LIN {X 0,Y 224.988,Z 280.423,A -85,B 0,C 180,E1 -22090.658,E2 -22090.658} C_VEL
LIN {X 0,Y 227.045,Z 246.583,A -85,B 0,C 180,E1 -22091.716,E2 -22091.716} C_VEL
LIN {X 0,Y 226.588,Z 244.432,A -85,B 0,C 180,E1 -22091.955,E2 -22091.955} C_VEL
LIN {X 0,Y 221.706,Z 232.717,A -85,B 0,C 180,E1 -22094.047,E2 -22094.047} C_VEL
LIN {X 0,Y 216.446,Z 222.08,A -85,B 0,C 180,E1 -22096.416,E2 -22096.416} C_VEL
LIN {X 0,Y 211.273,Z 212.801,A -85,B 0,C 180,E1 -22098.988,E2 -22098.988} C_VEL
LIN {X 0,Y 207.639,Z 206.885,A -85,B 0,C 180,E1 -22100.948,E2 -22100.948} C_VEL
LIN {X 0,Y 204.559,Z 201.986,A -85,B 0,C 180,E1 -22102.75,E2 -22102.75} C_VEL
LIN {X 0,Y 200.929,Z 196.512,A -85,B 0,C 180,E1 -22105.098,E2 -22105.098} C_VEL
LIN {X 0,Y 196.507,Z 190.274,A -85,B 0,C 180,E1 -22108.383,E2 -22108.383} C_VEL
LIN {X 0,Y 192.458,Z 184.954,A -85,B 0,C 180,E1 -22111.954,E2 -22111.954} C_VEL
LIN {X 0,Y 191.731,Z 183.77,A -85,B 0,C 180,E1 -22112.728,E2 -22112.728} C_VEL
LIN {X 0,Y 188.179,Z 179.993,A -85,B 0,C 180,E1 -22116.911,E2 -22116.911} C_VEL
LIN {X 0,Y 186.22,Z 177.647,A -85,B 0,C 180,E1 -22119.999,E2 -22119.999} C_VEL
LIN {X 0,Y 185.766,Z 176.032,A -85,B 0,C 180,E1 -22121.256,E2 -22121.256} C_VEL
LIN {X 0,Y 185.661,Z 175.348,A -85,B 0,C 180,E1 -22123.505,E2 -22123.505} C_VEL
LIN {X 0,Y 185.889,Z 175.33,A -85,B 0,C 180,E1 -22129.418,E2 -22129.418} C_VEL
LIN {X 0,Y 185.931,Z 175.314,A -85,B 0,C 180,E1 -22133.488,E2 -22133.488} C_VEL
LIN {X 0,Y 186.178,Z 175.278,A -85,B 0,C 180,E1 -22137.835,E2 -22137.835} C_VEL
LIN {X 0,Y 186.347,Z 175.263,A -85,B 0,C 180,E1 -22140.269,E2 -22140.269} C_VEL
LIN {X 0,Y 186.866,Z 177.432,A -85,B 0,C 180,E1 -22141.48,E2 -22141.48} C_VEL
LIN {X 0,Y 188.498,Z 179.95,A -85,B 0,C 180,E1 -22144.008,E2 -22144.008} C_VEL
LIN {X 0,Y 191.327,Z 181.512,A -85,B 0,C 180,E1 -22147.166,E2 -22147.166} C_VEL
LIN {X 0,Y 192.658,Z 184.369,A -85,B 0,C 180,E1 -22148.694,E2 -22148.694} C_VEL
LIN {X 0,Y 195.421,Z 186.847,A -85,B 0,C 180,E1 -22151.079,E2 -22151.079} C_VEL
LIN {X 0,Y 196.081,Z 187.718,A -85,B 0,C 180,E1 -22151.63,E2 -22151.63} C_VEL
LIN {X 0,Y 198.151,Z 190.841,A -85,B 0,C 180,E1 -22153.295,E2 -22153.295} C_VEL
LIN {X 0,Y 200.301,Z 192.877,A -85,B 0,C 180,E1 -22154.785,E2 -22154.785} C_VEL
LIN {X 0,Y 202.888,Z 196.511,A -85,B 0,C 180,E1 -22156.531,E2 -22156.531} C_VEL
LIN {X 0,Y 204.322,Z 198.272,A -85,B 0,C 180,E1 -22157.411,E2 -22157.411} C_VEL
LIN {X 0,Y 207.184,Z 201.939,A -85,B 0,C 180,E1 -22159.055,E2 -22159.055} C_VEL
LIN {X 0,Y 211.633,Z 208.287,A -85,B 0,C 180,E1 -22161.424,E2 -22161.424} C_VEL
LIN {X 0,Y 216.087,Z 214.791,A -85,B 0,C 180,E1 -22163.574,E2 -22163.574} C_VEL
LIN {X 0,Y 221.021,Z 223.069,A -85,B 0,C 180,E1 -22165.767,E2 -22165.767} C_VEL
LIN {X 0,Y 226.41,Z 233.873,A -85,B 0,C 180,E1 -22168.017,E2 -22168.017} C_VEL
LIN {X 0,Y 227.763,Z 236.952,A -85,B 0,C 180,E1 -22168.568,E2 -22168.568} C_VEL
LIN {X 0,Y 224.854,Z 278.71,A -85,B 0,C 180,E1 -22169.862,E2 -22169.862} C_VEL
LIN {X 0,Y 222.95,Z 292.239,A -85,B 0,C 180,E1 -22170.585,E2 -22170.585} C_VEL
LIN {X 0,Y 220.678,Z 304.196,A -85,B 0,C 180,E1 -22171.579,E2 -22171.579} C_VEL
LIN {X 0,Y 217.56,Z 315.965,A -85,B 0,C 180,E1 -22172.871,E2 -22172.871} C_VEL
LIN {X 0,Y 214.251,Z 326.305,A -85,B 0,C 180,E1 -22174.361,E2 -22174.361} C_VEL
LIN {X 0,Y 210.299,Z 336.7,A -85,B 0,C 180,E1 -22176.27,E2 -22176.27} C_VEL
LIN {X 0,Y 206.292,Z 345.823,A -85,B 0,C 180,E1 -22178.411,E2 -22178.411} C_VEL
LIN {X 0,Y 201.831,Z 354.704,A -85,B 0,C 180,E1 -22181.104,E2 -22181.104} C_VEL
LIN {X 0,Y 197.677,Z 362.007,A -85,B 0,C 180,E1 -22183.95,E2 -22183.95} C_VEL
LIN {X 0,Y 194.468,Z 367.315,A -85,B 0,C 180,E1 -22186.634,E2 -22186.634} C_VEL
LIN {X 0,Y 191.099,Z 372.35,A -85,B 0,C 180,E1 -22189.941,E2 -22189.941} C_VEL
LIN {X 0,Y 188.379,Z 376.088,A -85,B 0,C 180,E1 -22193.35,E2 -22193.35} C_VEL
LIN {X 0,Y 186.697,Z 378.058,A -85,B 0,C 180,E1 -22195.909,E2 -22195.909} C_VEL
LIN {X 0,Y 185.598,Z 379.226,A -85,B 0,C 180,E1 -22197.986,E2 -22197.986} C_VEL
LIN {X 0,Y 184.271,Z 380.301,A -85,B 0,C 180,E1 -22201.305,E2 -22201.305} C_VEL
LIN {X 0,Y 183.319,Z 380.428,A -85,B 0,C 180,E1 -22205.058,E2 -22205.058} C_VEL
LIN {X 0,Y 183.017,Z 379.943,A -85,B 0,C 180,E1 -22207.418,E2 -22207.418} C_VEL
LIN {X 0,Y 182.831,Z 378.973,A -85,B 0,C 180,E1 -22209.76,E2 -22209.76} C_VEL
LIN {X 0,Y 183.023,Z 376.309,A -85,B 0,C 180,E1 -22213.732,E2 -22213.732} C_VEL
LIN {X 0,Y 183.704,Z 372.053,A -85,B 0,C 180,E1 -22217.854,E2 -22217.854} C_VEL
LIN {X 0,Y 184.693,Z 366.57,A -85,B 0,C 180,E1 -22221.625,E2 -22221.625} C_VEL
LIN {X 0,Y 186.106,Z 359.926,A -85,B 0,C 180,E1 -22225.126,E2 -22225.126} C_VEL
LIN {X 0,Y 187.845,Z 352.004,A -85,B 0,C 180,E1 -22228.392,E2 -22228.392} C_VEL
LIN {X 0,Y 189.79,Z 343.547,A -85,B 0,C 180,E1 -22231.151,E2 -22231.151} C_VEL
LIN {X 0,Y 192.004,Z 333.872,A -85,B 0,C 180,E1 -22233.673,E2 -22233.673} C_VEL
LIN {X 0,Y 194.19,Z 322.773,A -85,B 0,C 180,E1 -22235.973,E2 -22235.973} C_VEL
LIN {X 0,Y 196.122,Z 311.841,A -85,B 0,C 180,E1 -22237.723,E2 -22237.723} C_VEL
LIN {X 0,Y 197.792,Z 299.873,A -85,B 0,C 180,E1 -22239.201,E2 -22239.201} C_VEL
LIN {X 0,Y 199.172,Z 286.973,A -85,B 0,C 180,E1 -22240.355,E2 -22240.355} C_VEL
LIN {X 0,Y 200.126,Z 274.306,A -85,B 0,C 180,E1 -22241.074,E2 -22241.074} C_VEL
LIN {X 0,Y 202.77,Z 214.463,A -85,B 0,C 180,E1 -22243.143,E2 -22243.143} C_VEL
LIN {X 0,Y 198.505,Z 201.646,A -85,B 0,C 180,E1 -22244.291,E2 -22244.291} C_VEL
LIN {X 0,Y 190.934,Z 186.085,A -85,B 0,C 180,E1 -22246.169,E2 -22246.169} C_VEL
LIN {X 0,Y 186.573,Z 178.087,A -85,B 0,C 180,E1 -22247.29,E2 -22247.29} C_VEL
LIN {X 0,Y 185.642,Z 175.362,A -85,B 0,C 180,E1 -22247.63,E2 -22247.63} C_VEL
LIN {X 0,Y 185.535,Z 175.354,A -85,B 0,C 180,E1 -22252.26,E2 -22252.26} C_VEL
LIN {X 0,Y 185.485,Z 175.339,A -85,B 0,C 180,E1 -22257.045,E2 -22257.045} C_VEL
LIN {X 0,Y 185.528,Z 175.375,A -85,B 0,C 180,E1 -22262.029,E2 -22262.029} C_VEL
LIN {X 0,Y 185.497,Z 175.361,A -85,B 0,C 180,E1 -22267.316,E2 -22267.316} C_VEL
LIN {X 0,Y 185.459,Z 175.383,A -85,B 0,C 180,E1 -22270.722,E2 -22270.722} C_VEL
LIN {X 0,Y 185.453,Z 175.353,A -85,B 0,C 180,E1 -22276.058,E2 -22276.058} C_VEL
LIN {X 0,Y 185.455,Z 175.373,A -85,B 0,C 180,E1 -22279.894,E2 -22279.894} C_VEL
LIN {X 0,Y 185.5,Z 175.378,A -85,B 0,C 180,E1 -22282.715,E2 -22282.715} C_VEL
LIN {X 0,Y 185.531,Z 175.345,A -85,B 0,C 180,E1 -22287.974,E2 -22287.974} C_VEL
LIN {X 0,Y 185.547,Z 175.327,A -85,B 0,C 180,E1 -22290.597,E2 -22290.597} C_VEL
LIN {X 0,Y 185.545,Z 175.365,A -85,B 0,C 180,E1 -22295.378,E2 -22295.378} C_VEL
LIN {X 0,Y 185.626,Z 175.356,A -85,B 0,C 180,E1 -22301.18,E2 -22301.18} C_VEL
LIN {X 0,Y 185.698,Z 175.353,A -85,B 0,C 180,E1 -22306.876,E2 -22306.876} C_VEL
LIN {X 0,Y 185.975,Z 175.306,A -85,B 0,C 180,E1 -22311.307,E2 -22311.307} C_VEL
LIN {X 0,Y 186.177,Z 175.29,A -85,B 0,C 180,E1 -22317.838,E2 -22317.838} C_VEL
LIN {X 0,Y 186.383,Z 175.258,A -85,B 0,C 180,E1 -22320.001,E2 -22320.001} C_VEL
LIN {X 0,Y 185.888,Z 175.331,A -85,B 0,C 180,E1 -22324.338,E2 -22324.338} C_VEL
LIN {X 0,Y 185.978,Z 175.309,A -85,B 0,C 180,E1 -22328.695,E2 -22328.695} C_VEL
LIN {X 0,Y 185.711,Z 175.354,A -85,B 0,C 180,E1 -22333.125,E2 -22333.125} C_VEL
LIN {X 0,Y 185.629,Z 175.361,A -85,B 0,C 180,E1 -22338.822,E2 -22338.822} C_VEL
LIN {X 0,Y 185.582,Z 175.368,A -85,B 0,C 180,E1 -22344.647,E2 -22344.647} C_VEL
LIN {X 0,Y 185.548,Z 175.372,A -85,B 0,C 180,E1 -22349.5,E2 -22349.5} C_VEL
LIN {X 0,Y 185.501,Z 175.379,A -85,B 0,C 180,E1 -22354.633,E2 -22354.633} C_VEL
LIN {X 0,Y 185.503,Z 175.38,A -85,B 0,C 180,E1 -22357.315,E2 -22357.315} C_VEL
LIN {X 0,Y 185.465,Z 175.387,A -85,B 0,C 180,E1 -22360.721,E2 -22360.721} C_VEL
LIN {X 0,Y 185.46,Z 175.388,A -85,B 0,C 180,E1 -22366.056,E2 -22366.056} C_VEL
LIN {X 0,Y 185.485,Z 175.438,A -85,B 0,C 180,E1 -22369.465,E2 -22369.465} C_VEL
LIN {X 0,Y 186.858,Z 180.956,A -85,B 0,C 180,E1 -22372.376,E2 -22372.376} C_VEL
LIN {X 0,Y 194.383,Z 199.087,A -85,B 0,C 180,E1 -22374.442,E2 -22374.442} C_VEL
LIN {X 0,Y 198.947,Z 211.96,A -85,B 0,C 180,E1 -22375.683,E2 -22375.683} C_VEL
LIN {X 0,Y 201.858,Z 239.357,A -85,B 0,C 180,E1 -22377.211,E2 -22377.211} C_VEL
LIN {X 0,Y 201.332,Z 253.298,A -85,B 0,C 180,E1 -22377.698,E2 -22377.698} C_VEL
LIN {X 0,Y 200.535,Z 259.13,A -85,B 0,C 180,E1 -22377.822,E2 -22377.822} C_VEL
LIN {X 0,Y 194.503,Z 278.032,A -85,B 0,C 180,E1 -22377.768,E2 -22377.768} C_VEL
LIN {X 0,Y 193.57,Z 283.859,A -85,B 0,C 180,E1 -22377.897,E2 -22377.897} C_VEL
LIN {X 0,Y 192.561,Z 297.296,A -85,B 0,C 180,E1 -22378.585,E2 -22378.585} C_VEL
LIN {X 0,Y 191.136,Z 309.973,A -85,B 0,C 180,E1 -22379.629,E2 -22379.629} C_VEL
LIN {X 0,Y 189.486,Z 320.811,A -85,B 0,C 180,E1 -22380.869,E2 -22380.869} C_VEL
LIN {X 0,Y 187.207,Z 332.465,A -85,B 0,C 180,E1 -22382.62,E2 -22382.62} C_VEL
LIN {X 0,Y 185.011,Z 343.062,A -85,B 0,C 180,E1 -22384.7,E2 -22384.7} C_VEL
LIN {X 0,Y 183.118,Z 351.772,A -85,B 0,C 180,E1 -22386.834,E2 -22386.834} C_VEL
LIN {X 0,Y 181.173,Z 359.673,A -85,B 0,C 180,E1 -22389.181,E2 -22389.181} C_VEL
LIN {X 0,Y 179.327,Z 368.161,A -85,B 0,C 180,E1 -22392.318,E2 -22392.318} C_VEL
LIN {X 0,Y 177.69,Z 375.411,A -85,B 0,C 180,E1 -22395.688,E2 -22395.688} C_VEL
LIN {X 0,Y 176.878,Z 380.303,A -85,B 0,C 180,E1 -22398.54,E2 -22398.54} C_VEL
LIN {X 0,Y 176.316,Z 385.025,A -85,B 0,C 180,E1 -22401.98,E2 -22401.98} C_VEL
LIN {X 0,Y 176.072,Z 388.591,A -85,B 0,C 180,E1 -22405.421,E2 -22405.421} C_VEL
LIN {X 0,Y 176.111,Z 390.397,A -85,B 0,C 180,E1 -22407.712,E2 -22407.712} C_VEL
LIN {X 0,Y 176.263,Z 391.74,A -85,B 0,C 180,E1 -22410,E2 -22410} C_VEL
LIN {X 0,Y 175.995,Z 392.946,A -85,B 0,C 180,E1 -22413.301,E2 -22413.301} C_VEL
LIN {X 0,Y 176.136,Z 393.318,A -85,B 0,C 180,E1 -22416.875,E2 -22416.875} C_VEL
LIN {X 0,Y 176.991,Z 392.371,A -85,B 0,C 180,E1 -22421.451,E2 -22421.451} C_VEL
LIN {X 0,Y 178.807,Z 389.906,A -85,B 0,C 180,E1 -22425.97,E2 -22425.97} C_VEL
LIN {X 0,Y 181.042,Z 386.95,A -85,B 0,C 180,E1 -22429.267,E2 -22429.267} C_VEL
LIN {X 0,Y 183.803,Z 382.992,A -85,B 0,C 180,E1 -22432.48,E2 -22432.48} C_VEL
LIN {X 0,Y 187.606,Z 377.012,A -85,B 0,C 180,E1 -22436.097,E2 -22436.097} C_VEL
LIN {X 0,Y 191.627,Z 370.438,A -85,B 0,C 180,E1 -22439.075,E2 -22439.075} C_VEL
LIN {X 0,Y 196.24,Z 362.341,A -85,B 0,C 180,E1 -22441.887,E2 -22441.887} C_VEL
LIN {X 0,Y 200.441,Z 354.106,A -85,B 0,C 180,E1 -22444.125,E2 -22444.125} C_VEL
LIN {X 0,Y 204.875,Z 344.085,A -85,B 0,C 180,E1 -22446.281,E2 -22446.281} C_VEL
LIN {X 0,Y 209.3,Z 332.76,A -85,B 0,C 180,E1 -22448.098,E2 -22448.098} C_VEL
LIN {X 0,Y 212.933,Z 321.686,A -85,B 0,C 180,E1 -22449.447,E2 -22449.447} C_VEL
LIN {X 0,Y 216.119,Z 309.391,A -85,B 0,C 180,E1 -22450.57,E2 -22450.57} C_VEL
LIN {X 0,Y 218.681,Z 296.076,A -85,B 0,C 180,E1 -22451.389,E2 -22451.389} C_VEL
LIN {X 0,Y 220.109,Z 282.961,A -85,B 0,C 180,E1 -22451.946,E2 -22451.946} C_VEL
LIN {X 0,Y 222.352,Z 248.258,A -85,B 0,C 180,E1 -22453.035,E2 -22453.035} C_VEL
LIN {X 0,Y 217.805,Z 237.081,A -85,B 0,C 180,E1 -22455.103,E2 -22455.103} C_VEL
LIN {X 0,Y 212.92,Z 226.864,A -85,B 0,C 180,E1 -22457.462,E2 -22457.462} C_VEL
LIN {X 0,Y 207.797,Z 217.518,A -85,B 0,C 180,E1 -22460.164,E2 -22460.164} C_VEL
LIN {X 0,Y 204.933,Z 212.689,A -85,B 0,C 180,E1 -22461.804,E2 -22461.804} C_VEL
LIN {X 0,Y 201.974,Z 207.827,A -85,B 0,C 180,E1 -22463.63,E2 -22463.63} C_VEL
LIN {X 0,Y 198.451,Z 202.392,A -85,B 0,C 180,E1 -22466.062,E2 -22466.062} C_VEL
LIN {X 0,Y 194.634,Z 196.721,A -85,B 0,C 180,E1 -22469.061,E2 -22469.061} C_VEL
LIN {X 0,Y 190.786,Z 191.474,A -85,B 0,C 180,E1 -22472.647,E2 -22472.647} C_VEL
LIN {X 0,Y 190.11,Z 190.384,A -85,B 0,C 180,E1 -22473.405,E2 -22473.405} C_VEL
LIN {X 0,Y 187.089,Z 186.979,A -85,B 0,C 180,E1 -22477.121,E2 -22477.121} C_VEL
LIN {X 0,Y 185.029,Z 184.475,A -85,B 0,C 180,E1 -22480.49,E2 -22480.49} C_VEL
LIN {X 0,Y 184.467,Z 182.792,A -85,B 0,C 180,E1 -22481.927,E2 -22481.927} C_VEL
LIN {X 0,Y 183.951,Z 182.236,A -85,B 0,C 180,E1 -22483.233,E2 -22483.233} C_VEL
LIN {X 0,Y 182.575,Z 181.546,A -85,B 0,C 180,E1 -22491.141,E2 -22491.141} C_VEL
LIN {X 0,Y 185.096,Z 182.442,A -85,B 0,C 180,E1 -22499.727,E2 -22499.727} C_VEL
LIN {X 0,Y 186.058,Z 185.122,A -85,B 0,C 180,E1 -22501.758,E2 -22501.758} C_VEL
LIN {X 0,Y 187.781,Z 187.248,A -85,B 0,C 180,E1 -22504.292,E2 -22504.292} C_VEL
LIN {X 0,Y 189.795,Z 188.45,A -85,B 0,C 180,E1 -22506.588,E2 -22506.588} C_VEL
LIN {X 0,Y 191.416,Z 191.422,A -85,B 0,C 180,E1 -22508.444,E2 -22508.444} C_VEL
LIN {X 0,Y 194.088,Z 193.996,A -85,B 0,C 180,E1 -22510.826,E2 -22510.826} C_VEL
LIN {X 0,Y 196.277,Z 197.335,A -85,B 0,C 180,E1 -22512.668,E2 -22512.668} C_VEL
LIN {X 0,Y 198.274,Z 199.379,A -85,B 0,C 180,E1 -22514.12,E2 -22514.12} C_VEL
LIN {X 0,Y 201.043,Z 203.14,A -85,B 0,C 180,E1 -22516.043,E2 -22516.043} C_VEL
LIN {X 0,Y 205.642,Z 209.545,A -85,B 0,C 180,E1 -22518.862,E2 -22518.862} C_VEL
LIN {X 0,Y 210.313,Z 216.136,A -85,B 0,C 180,E1 -22521.373,E2 -22521.373} C_VEL
LIN {X 0,Y 215.716,Z 224.86,A -85,B 0,C 180,E1 -22524.023,E2 -22524.023} C_VEL
LIN {X 0,Y 220.738,Z 234.637,A -85,B 0,C 180,E1 -22526.291,E2 -22526.291} C_VEL
LIN {X 0,Y 222.942,Z 239.558,A -85,B 0,C 180,E1 -22527.249,E2 -22527.249} C_VEL
LIN {X 0,Y 220.186,Z 278.627,A -85,B 0,C 180,E1 -22528.489,E2 -22528.489} C_VEL
LIN {X 0,Y 218.152,Z 292.57,A -85,B 0,C 180,E1 -22529.233,E2 -22529.233} C_VEL
LIN {X 0,Y 215.662,Z 304.983,A -85,B 0,C 180,E1 -22530.279,E2 -22530.279} C_VEL
LIN {X 0,Y 212.329,Z 316.934,A -85,B 0,C 180,E1 -22531.616,E2 -22531.616} C_VEL
LIN {X 0,Y 208.334,Z 328.745,A -85,B 0,C 180,E1 -22533.392,E2 -22533.392} C_VEL
LIN {X 0,Y 204.57,Z 337.95,A -85,B 0,C 180,E1 -22535.165,E2 -22535.165} C_VEL
LIN {X 0,Y 200.684,Z 346.296,A -85,B 0,C 180,E1 -22537.183,E2 -22537.183} C_VEL
LIN {X 0,Y 196.465,Z 354.302,A -85,B 0,C 180,E1 -22539.625,E2 -22539.625} C_VEL
LIN {X 0,Y 191.659,Z 362.392,A -85,B 0,C 180,E1 -22542.829,E2 -22542.829} C_VEL
LIN {X 0,Y 187.604,Z 368.614,A -85,B 0,C 180,E1 -22546.128,E2 -22546.128} C_VEL
LIN {X 0,Y 183.854,Z 373.726,A -85,B 0,C 180,E1 -22549.862,E2 -22549.862} C_VEL
LIN {X 0,Y 182.192,Z 375.832,A -85,B 0,C 180,E1 -22551.889,E2 -22551.889} C_VEL
LIN {X 0,Y 180.028,Z 378.307,A -85,B 0,C 180,E1 -22555.063,E2 -22555.063} C_VEL
LIN {X 0,Y 177.951,Z 380.196,A -85,B 0,C 180,E1 -22559.108,E2 -22559.108} C_VEL
LIN {X 0,Y 177.067,Z 380.717,A -85,B 0,C 180,E1 -22561.557,E2 -22561.557} C_VEL
LIN {X 0,Y 176.432,Z 380.743,A -85,B 0,C 180,E1 -22564.013,E2 -22564.013} C_VEL
LIN {X 0,Y 175.997,Z 380.293,A -85,B 0,C 180,E1 -22566.697,E2 -22566.697} C_VEL
LIN {X 0,Y 175.767,Z 379.517,A -85,B 0,C 180,E1 -22568.909,E2 -22568.909} C_VEL
LIN {X 0,Y 175.743,Z 378.198,A -85,B 0,C 180,E1 -22571.342,E2 -22571.342} C_VEL
LIN {X 0,Y 176.063,Z 375.392,A -85,B 0,C 180,E1 -22574.962,E2 -22574.962} C_VEL
LIN {X 0,Y 176.766,Z 371.503,A -85,B 0,C 180,E1 -22578.534,E2 -22578.534} C_VEL
LIN {X 0,Y 177.864,Z 365.816,A -85,B 0,C 180,E1 -22582.438,E2 -22582.438} C_VEL
LIN {X 0,Y 179.348,Z 358.888,A -85,B 0,C 180,E1 -22586.068,E2 -22586.068} C_VEL
LIN {X 0,Y 181.322,Z 350.599,A -85,B 0,C 180,E1 -22589.445,E2 -22589.445} C_VEL
LIN {X 0,Y 183.295,Z 342.136,A -85,B 0,C 180,E1 -22592.198,E2 -22592.198} C_VEL
LIN {X 0,Y 185.495,Z 332.853,A -85,B 0,C 180,E1 -22594.618,E2 -22594.618} C_VEL
LIN {X 0,Y 187.541,Z 322.786,A -85,B 0,C 180,E1 -22596.726,E2 -22596.726} C_VEL
LIN {X 0,Y 189.544,Z 311.799,A -85,B 0,C 180,E1 -22598.53,E2 -22598.53} C_VEL
LIN {X 0,Y 191.317,Z 299.731,A -85,B 0,C 180,E1 -22600.049,E2 -22600.049} C_VEL
LIN {X 0,Y 192.743,Z 286.623,A -85,B 0,C 180,E1 -22601.237,E2 -22601.237} C_VEL
LIN {X 0,Y 193.718,Z 274.13,A -85,B 0,C 180,E1 -22601.949,E2 -22601.949} C_VEL
LIN {X 0,Y 196.366,Z 215.943,A -85,B 0,C 180,E1 -22604.018,E2 -22604.018} C_VEL
LIN {X 0,Y 192.734,Z 204.849,A -85,B 0,C 180,E1 -22605.056,E2 -22605.056} C_VEL
LIN {X 0,Y 184.942,Z 188.795,A -85,B 0,C 180,E1 -22607.096,E2 -22607.096} C_VEL
LIN {X 0,Y 179.939,Z 179.621,A -85,B 0,C 180,E1 -22608.453,E2 -22608.453} C_VEL
LIN {X 0,Y 178.747,Z 177.144,A -85,B 0,C 180,E1 -22608.805,E2 -22608.805} C_VEL
LIN {X 0,Y 178.563,Z 176.242,A -85,B 0,C 180,E1 -22608.936,E2 -22608.936} C_VEL
LIN {X 0,Y 178.46,Z 176.202,A -85,B 0,C 180,E1 -22615.076,E2 -22615.076} C_VEL
LIN {X 0,Y 178.448,Z 176.254,A -85,B 0,C 180,E1 -22620.797,E2 -22620.797} C_VEL
LIN {X 0,Y 178.48,Z 176.243,A -85,B 0,C 180,E1 -22624.219,E2 -22624.219} C_VEL
LIN {X 0,Y 178.385,Z 176.259,A -85,B 0,C 180,E1 -22629.078,E2 -22629.078} C_VEL
LIN {X 0,Y 178.391,Z 176.262,A -85,B 0,C 180,E1 -22632.048,E2 -22632.048} C_VEL
LIN {X 0,Y 178.389,Z 176.238,A -85,B 0,C 180,E1 -22635.166,E2 -22635.166} C_VEL
LIN {X 0,Y 178.396,Z 176.239,A -85,B 0,C 180,E1 -22638.463,E2 -22638.463} C_VEL
LIN {X 0,Y 178.418,Z 176.258,A -85,B 0,C 180,E1 -22643.784,E2 -22643.784} C_VEL
LIN {X 0,Y 178.484,Z 176.235,A -85,B 0,C 180,E1 -22646.548,E2 -22646.548} C_VEL
LIN {X 0,Y 178.438,Z 176.216,A -85,B 0,C 180,E1 -22651.796,E2 -22651.796} C_VEL
LIN {X 0,Y 178.464,Z 176.253,A -85,B 0,C 180,E1 -22656.81,E2 -22656.81} C_VEL
LIN {X 0,Y 178.607,Z 176.228,A -85,B 0,C 180,E1 -22661.653,E2 -22661.653} C_VEL
LIN {X 0,Y 178.625,Z 176.236,A -85,B 0,C 180,E1 -22666.347,E2 -22666.347} C_VEL
LIN {X 0,Y 178.906,Z 176.186,A -85,B 0,C 180,E1 -22670.961,E2 -22670.961} C_VEL
LIN {X 0,Y 179.125,Z 176.168,A -85,B 0,C 180,E1 -22677.753,E2 -22677.753} C_VEL
LIN {X 0,Y 179.348,Z 176.134,A -85,B 0,C 180,E1 -22680.001,E2 -22680.001} C_VEL
LIN {X 0,Y 178.837,Z 176.209,A -85,B 0,C 180,E1 -22684.509,E2 -22684.509} C_VEL
LIN {X 0,Y 178.908,Z 176.19,A -85,B 0,C 180,E1 -22689.042,E2 -22689.042} C_VEL
LIN {X 0,Y 178.637,Z 176.231,A -85,B 0,C 180,E1 -22693.655,E2 -22693.655} C_VEL
LIN {X 0,Y 178.558,Z 176.243,A -85,B 0,C 180,E1 -22699.152,E2 -22699.152} C_VEL
LIN {X 0,Y 178.52,Z 176.247,A -85,B 0,C 180,E1 -22705.112,E2 -22705.112} C_VEL
LIN {X 0,Y 178.464,Z 176.255,A -85,B 0,C 180,E1 -22710.795,E2 -22710.795} C_VEL
LIN {X 0,Y 178.487,Z 176.252,A -85,B 0,C 180,E1 -22714.219,E2 -22714.219} C_VEL
LIN {X 0,Y 178.391,Z 176.268,A -85,B 0,C 180,E1 -22719.077,E2 -22719.077} C_VEL
LIN {X 0,Y 178.397,Z 176.267,A -85,B 0,C 180,E1 -22722.047,E2 -22722.047} C_VEL
LIN {X 0,Y 178.395,Z 176.268,A -85,B 0,C 180,E1 -22725.165,E2 -22725.165} C_VEL
LIN {X 0,Y 178.405,Z 176.296,A -85,B 0,C 180,E1 -22728.566,E2 -22728.566} C_VEL
LIN {X 0,Y 179.486,Z 180.614,A -85,B 0,C 180,E1 -22730.989,E2 -22730.989} C_VEL
LIN {X 0,Y 186.31,Z 196.313,A -85,B 0,C 180,E1 -22732.968,E2 -22732.968} C_VEL
LIN {X 0,Y 192.686,Z 213.811,A -85,B 0,C 180,E1 -22734.804,E2 -22734.804} C_VEL
LIN {X 0,Y 195.448,Z 240.415,A -85,B 0,C 180,E1 -22736.35,E2 -22736.35} C_VEL
LIN {X 0,Y 193.57,Z 283.859,A -85,B 0,C 180,E1 -22737.897,E2 -22737.897} C_VEL
LIN {X 0,Y 192.6,Z 289.657,A -85,B 0,C 180,E1 -22738.058,E2 -22738.058} C_VEL
LIN {X 0,Y 187.698,Z 302.596,A -85,B 0,C 180,E1 -22738.392,E2 -22738.392} C_VEL
LIN {X 0,Y 184.658,Z 310.825,A -85,B 0,C 180,E1 -22738.886,E2 -22738.886} C_VEL
LIN {X 0,Y 184.019,Z 313.58,A -85,B 0,C 180,E1 -22739.164,E2 -22739.164} C_VEL
LIN {X 0,Y 182.229,Z 324.208,A -85,B 0,C 180,E1 -22740.545,E2 -22740.545} C_VEL
LIN {X 0,Y 179.897,Z 335.113,A -85,B 0,C 180,E1 -22742.359,E2 -22742.359} C_VEL
LIN {X 0,Y 177.638,Z 345.181,A -85,B 0,C 180,E1 -22744.516,E2 -22744.516} C_VEL
LIN {X 0,Y 175.582,Z 354.415,A -85,B 0,C 180,E1 -22747.019,E2 -22747.019} C_VEL
LIN {X 0,Y 174.234,Z 359.683,A -85,B 0,C 180,E1 -22748.713,E2 -22748.713} C_VEL
LIN {X 0,Y 172.212,Z 368.61,A -85,B 0,C 180,E1 -22752.177,E2 -22752.177} C_VEL
LIN {X 0,Y 170.543,Z 375.685,A -85,B 0,C 180,E1 -22755.684,E2 -22755.684} C_VEL
LIN {X 0,Y 169.633,Z 381.343,A -85,B 0,C 180,E1 -22759.255,E2 -22759.255} C_VEL
LIN {X 0,Y 169.15,Z 385.758,A -85,B 0,C 180,E1 -22762.839,E2 -22762.839} C_VEL
LIN {X 0,Y 169.004,Z 389.058,A -85,B 0,C 180,E1 -22766.424,E2 -22766.424} C_VEL
LIN {X 0,Y 169.182,Z 391.344,A -85,B 0,C 180,E1 -22770,E2 -22770} C_VEL
LIN {X 0,Y 168.932,Z 392.541,A -85,B 0,C 180,E1 -22773.16,E2 -22773.16} C_VEL
LIN {X 0,Y 169.088,Z 393.054,A -85,B 0,C 180,E1 -22777.163,E2 -22777.163} C_VEL
LIN {X 0,Y 170.022,Z 392.206,A -85,B 0,C 180,E1 -22781.927,E2 -22781.927} C_VEL
LIN {X 0,Y 171.965,Z 389.825,A -85,B 0,C 180,E1 -22786.623,E2 -22786.623} C_VEL
LIN {X 0,Y 174.348,Z 386.955,A -85,B 0,C 180,E1 -22790.037,E2 -22790.037} C_VEL
LIN {X 0,Y 177.258,Z 383.097,A -85,B 0,C 180,E1 -22793.358,E2 -22793.358} C_VEL
LIN {X 0,Y 181.129,Z 377.442,A -85,B 0,C 180,E1 -22796.991,E2 -22796.991} C_VEL
LIN {X 0,Y 185.48,Z 370.818,A -85,B 0,C 180,E1 -22800.136,E2 -22800.136} C_VEL
LIN {X 0,Y 190.284,Z 362.852,A -85,B 0,C 180,E1 -22803.009,E2 -22803.009} C_VEL
LIN {X 0,Y 194.628,Z 354.772,A -85,B 0,C 180,E1 -22805.293,E2 -22805.293} C_VEL
LIN {X 0,Y 199.244,Z 344.963,A -85,B 0,C 180,E1 -22807.478,E2 -22807.478} C_VEL
LIN {X 0,Y 203.811,Z 333.971,A -85,B 0,C 180,E1 -22809.318,E2 -22809.318} C_VEL
LIN {X 0,Y 207.561,Z 323.244,A -85,B 0,C 180,E1 -22810.678,E2 -22810.678} C_VEL
LIN {X 0,Y 210.838,Z 311.497,A -85,B 0,C 180,E1 -22811.811,E2 -22811.811} C_VEL
LIN {X 0,Y 213.682,Z 298.309,A -85,B 0,C 180,E1 -22812.69,E2 -22812.69} C_VEL
LIN {X 0,Y 215.364,Z 284.732,A -85,B 0,C 180,E1 -22813.311,E2 -22813.311} C_VEL
LIN {X 0,Y 217.736,Z 250.798,A -85,B 0,C 180,E1 -22814.379,E2 -22814.379} C_VEL
LIN {X 0,Y 213.121,Z 239.421,A -85,B 0,C 180,E1 -22816.638,E2 -22816.638} C_VEL
LIN {X 0,Y 207.823,Z 228.417,A -85,B 0,C 180,E1 -22819.438,E2 -22819.438} C_VEL
LIN {X 0,Y 202.713,Z 219.168,A -85,B 0,C 180,E1 -22822.416,E2 -22822.416} C_VEL
LIN {X 0,Y 199.323,Z 213.462,A -85,B 0,C 180,E1 -22824.635,E2 -22824.635} C_VEL
LIN {X 0,Y 196.274,Z 208.571,A -85,B 0,C 180,E1 -22826.866,E2 -22826.866} C_VEL
LIN {X 0,Y 192.627,Z 202.971,A -85,B 0,C 180,E1 -22829.894,E2 -22829.894} C_VEL
LIN {X 0,Y 189.026,Z 197.739,A -85,B 0,C 180,E1 -22833.501,E2 -22833.501} C_VEL
LIN {X 0,Y 186.054,Z 194.004,A -85,B 0,C 180,E1 -22837.26,E2 -22837.26} C_VEL
LIN {X 0,Y 183.882,Z 191.356,A -85,B 0,C 180,E1 -22840.922,E2 -22840.922} C_VEL
LIN {X 0,Y 183.357,Z 189.661,A -85,B 0,C 180,E1 -22842.403,E2 -22842.403} C_VEL
LIN {X 0,Y 182.298,Z 189.046,A -85,B 0,C 180,E1 -22845.486,E2 -22845.486} C_VEL
LIN {X 0,Y 181.674,Z 188.591,A -85,B 0,C 180,E1 -22851.097,E2 -22851.097} C_VEL
LIN {X 0,Y 183.902,Z 189.397,A -85,B 0,C 180,E1 -22859.178,E2 -22859.178} C_VEL
LIN {X 0,Y 185.348,Z 192.854,A -85,B 0,C 180,E1 -22862.172,E2 -22862.172} C_VEL
LIN {X 0,Y 187.299,Z 194.596,A -85,B 0,C 180,E1 -22864.842,E2 -22864.842} C_VEL
LIN {X 0,Y 188.243,Z 195.145,A -85,B 0,C 180,E1 -22865.925,E2 -22865.925} C_VEL
LIN {X 0,Y 190.059,Z 198.341,A -85,B 0,C 180,E1 -22868.069,E2 -22868.069} C_VEL
LIN {X 0,Y 192.327,Z 200.652,A -85,B 0,C 180,E1 -22870.193,E2 -22870.193} C_VEL
LIN {X 0,Y 194.757,Z 204.224,A -85,B 0,C 180,E1 -22872.292,E2 -22872.292} C_VEL
LIN {X 0,Y 196.375,Z 205.994,A -85,B 0,C 180,E1 -22873.516,E2 -22873.516} C_VEL
LIN {X 0,Y 199.905,Z 211.008,A -85,B 0,C 180,E1 -22876.039,E2 -22876.039} C_VEL
LIN {X 0,Y 203.442,Z 216.022,A -85,B 0,C 180,E1 -22878.266,E2 -22878.266} C_VEL
LIN {X 0,Y 207.885,Z 222.615,A -85,B 0,C 180,E1 -22880.758,E2 -22880.758} C_VEL
LIN {X 0,Y 212.651,Z 230.509,A -85,B 0,C 180,E1 -22883.2,E2 -22883.2} C_VEL
LIN {X 0,Y 217.665,Z 240.812,A -85,B 0,C 180,E1 -22885.606,E2 -22885.606} C_VEL
LIN {X 0,Y 218.359,Z 242.396,A -85,B 0,C 180,E1 -22885.924,E2 -22885.924} C_VEL
LIN {X 0,Y 215.537,Z 279.381,A -85,B 0,C 180,E1 -22887.091,E2 -22887.091} C_VEL
LIN {X 0,Y 213.524,Z 292.632,A -85,B 0,C 180,E1 -22887.801,E2 -22887.801} C_VEL
LIN {X 0,Y 211.021,Z 304.655,A -85,B 0,C 180,E1 -22888.797,E2 -22888.797} C_VEL
LIN {X 0,Y 207.589,Z 316.777,A -85,B 0,C 180,E1 -22890.158,E2 -22890.158} C_VEL
LIN {X 0,Y 203.654,Z 327.939,A -85,B 0,C 180,E1 -22891.81,E2 -22891.81} C_VEL
LIN {X 0,Y 199.04,Z 338.85,A -85,B 0,C 180,E1 -22893.927,E2 -22893.927} C_VEL
LIN {X 0,Y 194.243,Z 348.512,A -85,B 0,C 180,E1 -22896.386,E2 -22896.386} C_VEL
LIN {X 0,Y 189.675,Z 356.595,A -85,B 0,C 180,E1 -22899.041,E2 -22899.041} C_VEL
LIN {X 0,Y 184.937,Z 363.933,A -85,B 0,C 180,E1 -22902.18,E2 -22902.18} C_VEL
LIN {X 0,Y 180.753,Z 369.838,A -85,B 0,C 180,E1 -22905.583,E2 -22905.583} C_VEL
LIN {X 0,Y 177.479,Z 374.006,A -85,B 0,C 180,E1 -22908.795,E2 -22908.795} C_VEL
LIN {X 0,Y 174.28,Z 377.652,A -85,B 0,C 180,E1 -22912.779,E2 -22912.779} C_VEL
LIN {X 0,Y 172.714,Z 379.224,A -85,B 0,C 180,E1 -22915.272,E2 -22915.272} C_VEL
LIN {X 0,Y 170.492,Z 380.823,A -85,B 0,C 180,E1 -22919.955,E2 -22919.955} C_VEL
LIN {X 0,Y 169.569,Z 381.06,A -85,B 0,C 180,E1 -22922.877,E2 -22922.877} C_VEL
LIN {X 0,Y 168.948,Z 380.566,A -85,B 0,C 180,E1 -22926.227,E2 -22926.227} C_VEL
LIN {X 0,Y 168.619,Z 378.823,A -85,B 0,C 180,E1 -22930.523,E2 -22930.523} C_VEL
LIN {X 0,Y 168.781,Z 376.98,A -85,B 0,C 180,E1 -22933.273,E2 -22933.273} C_VEL
LIN {X 0,Y 169.28,Z 373.794,A -85,B 0,C 180,E1 -22936.801,E2 -22936.801} C_VEL
LIN {X 0,Y 170.127,Z 369.321,A -85,B 0,C 180,E1 -22940.489,E2 -22940.489} C_VEL
LIN {X 0,Y 171.351,Z 363.616,A -85,B 0,C 180,E1 -22944.115,E2 -22944.115} C_VEL
LIN {X 0,Y 173.045,Z 356.485,A -85,B 0,C 180,E1 -22947.673,E2 -22947.673} C_VEL
LIN {X 0,Y 174.927,Z 349.007,A -85,B 0,C 180,E1 -22950.633,E2 -22950.633} C_VEL
LIN {X 0,Y 177.297,Z 339.29,A -85,B 0,C 180,E1 -22953.694,E2 -22953.694} C_VEL
LIN {X 0,Y 179.566,Z 329.345,A -85,B 0,C 180,E1 -22956.179,E2 -22956.179} C_VEL
LIN {X 0,Y 181.811,Z 318.397,A -85,B 0,C 180,E1 -22958.335,E2 -22958.335} C_VEL
LIN {X 0,Y 183.591,Z 308.122,A -85,B 0,C 180,E1 -22959.92,E2 -22959.92} C_VEL
LIN {X 0,Y 185.379,Z 295.846,A -85,B 0,C 180,E1 -22961.343,E2 -22961.343} C_VEL
LIN {X 0,Y 186.684,Z 282.619,A -85,B 0,C 180,E1 -22962.433,E2 -22962.433} C_VEL
LIN {X 0,Y 187.545,Z 269.477,A -85,B 0,C 180,E1 -22963.072,E2 -22963.072} C_VEL
LIN {X 0,Y 190.035,Z 217.332,A -85,B 0,C 180,E1 -22964.951,E2 -22964.951} C_VEL
LIN {X 0,Y 186.878,Z 207.776,A -85,B 0,C 180,E1 -22965.902,E2 -22965.902} C_VEL
LIN {X 0,Y 178.42,Z 190.405,A -85,B 0,C 180,E1 -22968.235,E2 -22968.235} C_VEL
LIN {X 0,Y 173.012,Z 180.75,A -85,B 0,C 180,E1 -22969.804,E2 -22969.804} C_VEL
LIN {X 0,Y 171.596,Z 177.916,A -85,B 0,C 180,E1 -22970.251,E2 -22970.251} C_VEL
LIN {X 0,Y 171.45,Z 177.128,A -85,B 0,C 180,E1 -22970.358,E2 -22970.358} C_VEL
LIN {X 0,Y 171.398,Z 177.079,A -85,B 0,C 180,E1 -22975.569,E2 -22975.569} C_VEL
LIN {X 0,Y 171.403,Z 177.131,A -85,B 0,C 180,E1 -22980.567,E2 -22980.567} C_VEL
LIN {X 0,Y 171.39,Z 177.117,A -85,B 0,C 180,E1 -22985.036,E2 -22985.036} C_VEL
LIN {X 0,Y 171.341,Z 177.135,A -85,B 0,C 180,E1 -22988.802,E2 -22988.802} C_VEL
LIN {X 0,Y 171.317,Z 177.126,A -85,B 0,C 180,E1 -22994.22,E2 -22994.22} C_VEL
LIN {X 0,Y 171.328,Z 177.121,A -85,B 0,C 180,E1 -22998.981,E2 -22998.981} C_VEL
LIN {X 0,Y 171.359,Z 177.136,A -85,B 0,C 180,E1 -23002.035,E2 -23002.035} C_VEL
LIN {X 0,Y 171.397,Z 177.127,A -85,B 0,C 180,E1 -23005.095,E2 -23005.095} C_VEL
LIN {X 0,Y 171.407,Z 177.083,A -85,B 0,C 180,E1 -23010.528,E2 -23010.528} C_VEL
LIN {X 0,Y 171.404,Z 177.127,A -85,B 0,C 180,E1 -23015.795,E2 -23015.795} C_VEL
LIN {X 0,Y 171.509,Z 177.114,A -85,B 0,C 180,E1 -23020.865,E2 -23020.865} C_VEL
LIN {X 0,Y 171.541,Z 177.116,A -85,B 0,C 180,E1 -23025.771,E2 -23025.771} C_VEL
LIN {X 0,Y 171.844,Z 177.066,A -85,B 0,C 180,E1 -23030.586,E2 -23030.586} C_VEL
LIN {X 0,Y 171.783,Z 177.088,A -85,B 0,C 180,E1 -23035.308,E2 -23035.308} C_VEL
LIN {X 0,Y 172.312,Z 177.01,A -85,B 0,C 180,E1 -23040.001,E2 -23040.001} C_VEL
LIN {X 0,Y 171.787,Z 177.087,A -85,B 0,C 180,E1 -23044.695,E2 -23044.695} C_VEL
LIN {X 0,Y 171.847,Z 177.071,A -85,B 0,C 180,E1 -23049.416,E2 -23049.416} C_VEL
LIN {X 0,Y 171.551,Z 177.112,A -85,B 0,C 180,E1 -23054.231,E2 -23054.231} C_VEL
LIN {X 0,Y 171.483,Z 177.126,A -85,B 0,C 180,E1 -23059.501,E2 -23059.501} C_VEL
LIN {X 0,Y 171.448,Z 177.128,A -85,B 0,C 180,E1 -23065.599,E2 -23065.599} C_VEL
LIN {X 0,Y 171.422,Z 177.131,A -85,B 0,C 180,E1 -23070.573,E2 -23070.573} C_VEL
LIN {X 0,Y 171.396,Z 177.138,A -85,B 0,C 180,E1 -23075.035,E2 -23075.035} C_VEL
LIN {X 0,Y 171.347,Z 177.146,A -85,B 0,C 180,E1 -23078.802,E2 -23078.802} C_VEL
LIN {X 0,Y 171.322,Z 177.149,A -85,B 0,C 180,E1 -23084.218,E2 -23084.218} C_VEL
LIN {X 0,Y 171.336,Z 177.146,A -85,B 0,C 180,E1 -23087.592,E2 -23087.592} C_VEL
LIN {X 0,Y 172.143,Z 180.386,A -85,B 0,C 180,E1 -23089.473,E2 -23089.473} C_VEL
LIN {X 0,Y 179.345,Z 196.319,A -85,B 0,C 180,E1 -23091.705,E2 -23091.705} C_VEL
LIN {X 0,Y 185.103,Z 211.559,A -85,B 0,C 180,E1 -23093.444,E2 -23093.444} C_VEL
LIN {X 0,Y 186.729,Z 216.868,A -85,B 0,C 180,E1 -23093.963,E2 -23093.963} C_VEL
LIN {X 0,Y 189.135,Z 240.036,A -85,B 0,C 180,E1 -23095.376,E2 -23095.376} C_VEL
LIN {X 0,Y 186.871,Z 289.382,A -85,B 0,C 180,E1 -23097.232,E2 -23097.232} C_VEL
LIN {X 0,Y 185.521,Z 302.928,A -85,B 0,C 180,E1 -23098.13,E2 -23098.13} C_VEL
LIN {X 0,Y 184.019,Z 313.58,A -85,B 0,C 180,E1 -23099.164,E2 -23099.164} C_VEL
LIN {X 0,Y 182.374,Z 319.005,A -85,B 0,C 180,E1 -23099.713,E2 -23099.713} C_VEL
LIN {X 0,Y 178.075,Z 327.54,A -85,B 0,C 180,E1 -23100.59,E2 -23100.59} C_VEL
LIN {X 0,Y 173.743,Z 335.696,A -85,B 0,C 180,E1 -23101.749,E2 -23101.749} C_VEL
LIN {X 0,Y 172.073,Z 340.516,A -85,B 0,C 180,E1 -23102.728,E2 -23102.728} C_VEL
LIN {X 0,Y 170,Z 349.318,A -85,B 0,C 180,E1 -23104.928,E2 -23104.928} C_VEL
LIN {X 0,Y 167.511,Z 358.611,A -85,B 0,C 180,E1 -23107.814,E2 -23107.814} C_VEL
LIN {X 0,Y 166.031,Z 364.905,A -85,B 0,C 180,E1 -23110.206,E2 -23110.206} C_VEL
LIN {X 0,Y 164.157,Z 372.673,A -85,B 0,C 180,E1 -23113.842,E2 -23113.842} C_VEL
LIN {X 0,Y 162.885,Z 378.893,A -85,B 0,C 180,E1 -23117.541,E2 -23117.541} C_VEL
LIN {X 0,Y 162.21,Z 383.808,A -85,B 0,C 180,E1 -23121.277,E2 -23121.277} C_VEL
LIN {X 0,Y 161.93,Z 387.554,A -85,B 0,C 180,E1 -23125.02,E2 -23125.02} C_VEL
LIN {X 0,Y 161.929,Z 389.47,A -85,B 0,C 180,E1 -23127.512,E2 -23127.512} C_VEL
LIN {X 0,Y 162.083,Z 390.946,A -85,B 0,C 180,E1 -23130,E2 -23130} C_VEL
LIN {X 0,Y 161.876,Z 392.11,A -85,B 0,C 180,E1 -23133.048,E2 -23133.048} C_VEL
LIN {X 0,Y 162.016,Z 392.772,A -85,B 0,C 180,E1 -23137.477,E2 -23137.477} C_VEL
LIN {X 0,Y 162.394,Z 392.617,A -85,B 0,C 180,E1 -23139.968,E2 -23139.968} C_VEL
LIN {X 0,Y 163.952,Z 391.09,A -85,B 0,C 180,E1 -23144.903,E2 -23144.903} C_VEL
LIN {X 0,Y 165.154,Z 389.754,A -85,B 0,C 180,E1 -23147.33,E2 -23147.33} C_VEL
LIN {X 0,Y 167.687,Z 386.973,A -85,B 0,C 180,E1 -23150.87,E2 -23150.87} C_VEL
LIN {X 0,Y 170.761,Z 383.208,A -85,B 0,C 180,E1 -23154.303,E2 -23154.303} C_VEL
LIN {X 0,Y 174.695,Z 377.852,A -85,B 0,C 180,E1 -23157.928,E2 -23157.928} C_VEL
LIN {X 0,Y 179.381,Z 371.183,A -85,B 0,C 180,E1 -23161.273,E2 -23161.273} C_VEL
LIN {X 0,Y 184.407,Z 363.363,A -85,B 0,C 180,E1 -23164.204,E2 -23164.204} C_VEL
LIN {X 0,Y 188.913,Z 355.435,A -85,B 0,C 180,E1 -23166.529,E2 -23166.529} C_VEL
LIN {X 0,Y 193.684,Z 345.813,A -85,B 0,C 180,E1 -23168.751,E2 -23168.751} C_VEL
LIN {X 0,Y 198.439,Z 335.128,A -85,B 0,C 180,E1 -23170.6,E2 -23170.6} C_VEL
LIN {X 0,Y 202.267,Z 324.794,A -85,B 0,C 180,E1 -23171.979,E2 -23171.979} C_VEL
LIN {X 0,Y 205.665,Z 313.553,A -85,B 0,C 180,E1 -23173.113,E2 -23173.113} C_VEL
LIN {X 0,Y 208.627,Z 300.952,A -85,B 0,C 180,E1 -23174.015,E2 -23174.015} C_VEL
LIN {X 0,Y 210.65,Z 287.567,A -85,B 0,C 180,E1 -23174.694,E2 -23174.694} C_VEL
LIN {X 0,Y 213.224,Z 253.314,A -85,B 0,C 180,E1 -23175.79,E2 -23175.79} C_VEL
LIN {X 0,Y 208.84,Z 242.448,A -85,B 0,C 180,E1 -23178.122,E2 -23178.122} C_VEL
LIN {X 0,Y 204.432,Z 233.132,A -85,B 0,C 180,E1 -23180.62,E2 -23180.62} C_VEL
LIN {X 0,Y 199.819,Z 224.53,A -85,B 0,C 180,E1 -23183.488,E2 -23183.488} C_VEL
LIN {X 0,Y 196.83,Z 219.267,A -85,B 0,C 180,E1 -23185.598,E2 -23185.598} C_VEL
LIN {X 0,Y 194.067,Z 214.66,A -85,B 0,C 180,E1 -23187.742,E2 -23187.742} C_VEL
LIN {X 0,Y 190.774,Z 209.365,A -85,B 0,C 180,E1 -23190.638,E2 -23190.638} C_VEL
LIN {X 0,Y 187.308,Z 204.014,A -85,B 0,C 180,E1 -23194.369,E2 -23194.369} C_VEL
LIN {X 0,Y 184.473,Z 200.592,A -85,B 0,C 180,E1 -23198.194,E2 -23198.194} C_VEL
LIN {X 0,Y 182.599,Z 197.811,A -85,B 0,C 180,E1 -23201.789,E2 -23201.789} C_VEL
LIN {X 0,Y 182.205,Z 196.453,A -85,B 0,C 180,E1 -23203.04,E2 -23203.04} C_VEL
LIN {X 0,Y 180.773,Z 195.637,A -85,B 0,C 180,E1 -23211.052,E2 -23211.052} C_VEL
LIN {X 0,Y 182.773,Z 196.413,A -85,B 0,C 180,E1 -23218.734,E2 -23218.734} C_VEL
LIN {X 0,Y 184.289,Z 199.891,A -85,B 0,C 180,E1 -23221.979,E2 -23221.979} C_VEL
LIN {X 0,Y 186.385,Z 201.666,A -85,B 0,C 180,E1 -23224.866,E2 -23224.866} C_VEL
LIN {X 0,Y 186.944,Z 202.287,A -85,B 0,C 180,E1 -23225.561,E2 -23225.561} C_VEL
LIN {X 0,Y 188.912,Z 205.449,A -85,B 0,C 180,E1 -23227.9,E2 -23227.9} C_VEL
LIN {X 0,Y 190.604,Z 207.28,A -85,B 0,C 180,E1 -23229.558,E2 -23229.558} C_VEL
LIN {X 0,Y 193.066,Z 210.886,A -85,B 0,C 180,E1 -23231.764,E2 -23231.764} C_VEL
LIN {X 0,Y 194.439,Z 212.527,A -85,B 0,C 180,E1 -23232.856,E2 -23232.856} C_VEL
LIN {X 0,Y 197.807,Z 217.453,A -85,B 0,C 180,E1 -23235.371,E2 -23235.371} C_VEL
LIN {X 0,Y 201.174,Z 222.362,A -85,B 0,C 180,E1 -23237.603,E2 -23237.603} C_VEL
LIN {X 0,Y 206.69,Z 230.933,A -85,B 0,C 180,E1 -23240.786,E2 -23240.786} C_VEL
LIN {X 0,Y 210.714,Z 238.283,A -85,B 0,C 180,E1 -23242.916,E2 -23242.916} C_VEL
LIN {X 0,Y 213.827,Z 245.119,A -85,B 0,C 180,E1 -23244.503,E2 -23244.503} C_VEL
LIN {X 0,Y 211.134,Z 279.347,A -85,B 0,C 180,E1 -23245.601,E2 -23245.601} C_VEL
LIN {X 0,Y 209.011,Z 292.876,A -85,B 0,C 180,E1 -23246.322,E2 -23246.322} C_VEL
LIN {X 0,Y 206.263,Z 305.452,A -85,B 0,C 180,E1 -23247.373,E2 -23247.373} C_VEL
LIN {X 0,Y 203.051,Z 316.471,A -85,B 0,C 180,E1 -23248.618,E2 -23248.618} C_VEL
LIN {X 0,Y 199.165,Z 327.147,A -85,B 0,C 180,E1 -23250.17,E2 -23250.17} C_VEL
LIN {X 0,Y 194.859,Z 337.152,A -85,B 0,C 180,E1 -23252.051,E2 -23252.051} C_VEL
LIN {X 0,Y 190.726,Z 345.469,A -85,B 0,C 180,E1 -23254.037,E2 -23254.037} C_VEL
LIN {X 0,Y 185.961,Z 353.883,A -85,B 0,C 180,E1 -23256.573,E2 -23256.573} C_VEL
LIN {X 0,Y 181.525,Z 360.806,A -85,B 0,C 180,E1 -23259.256,E2 -23259.256} C_VEL
LIN {X 0,Y 177.009,Z 367.121,A -85,B 0,C 180,E1 -23262.45,E2 -23262.45} C_VEL
LIN {X 0,Y 172.629,Z 372.613,A -85,B 0,C 180,E1 -23266.204,E2 -23266.204} C_VEL
LIN {X 0,Y 169.186,Z 376.485,A -85,B 0,C 180,E1 -23269.919,E2 -23269.919} C_VEL
LIN {X 0,Y 166.389,Z 379.173,A -85,B 0,C 180,E1 -23273.748,E2 -23273.748} C_VEL
LIN {X 0,Y 164.921,Z 380.362,A -85,B 0,C 180,E1 -23276.359,E2 -23276.359} C_VEL
LIN {X 0,Y 163.645,Z 381.09,A -85,B 0,C 180,E1 -23279.194,E2 -23279.194} C_VEL
LIN {X 0,Y 162.782,Z 381.319,A -85,B 0,C 180,E1 -23281.646,E2 -23281.646} C_VEL
LIN {X 0,Y 161.947,Z 380.842,A -85,B 0,C 180,E1 -23285.687,E2 -23285.687} C_VEL
LIN {X 0,Y 161.545,Z 379.381,A -85,B 0,C 180,E1 -23289.633,E2 -23289.633} C_VEL
LIN {X 0,Y 161.653,Z 377.302,A -85,B 0,C 180,E1 -23293.027,E2 -23293.027} C_VEL
LIN {X 0,Y 162.317,Z 373.342,A -85,B 0,C 180,E1 -23297.497,E2 -23297.497} C_VEL
LIN {X 0,Y 163.339,Z 368.109,A -85,B 0,C 180,E1 -23301.728,E2 -23301.728} C_VEL
LIN {X 0,Y 164.909,Z 361.553,A -85,B 0,C 180,E1 -23305.723,E2 -23305.723} C_VEL
LIN {X 0,Y 166.835,Z 353.844,A -85,B 0,C 180,E1 -23309.397,E2 -23309.397} C_VEL
LIN {X 0,Y 168.903,Z 345.946,A -85,B 0,C 180,E1 -23312.385,E2 -23312.385} C_VEL
LIN {X 0,Y 171.364,Z 336.266,A -85,B 0,C 180,E1 -23315.295,E2 -23315.295} C_VEL
LIN {X 0,Y 173.825,Z 325.515,A -85,B 0,C 180,E1 -23317.843,E2 -23317.843} C_VEL
LIN {X 0,Y 175.986,Z 315.121,A -85,B 0,C 180,E1 -23319.772,E2 -23319.772} C_VEL
LIN {X 0,Y 177.972,Z 302.876,A -85,B 0,C 180,E1 -23321.533,E2 -23321.533} C_VEL
LIN {X 0,Y 179.629,Z 289.978,A -85,B 0,C 180,E1 -23322.858,E2 -23322.858} C_VEL
LIN {X 0,Y 180.82,Z 277.19,A -85,B 0,C 180,E1 -23323.728,E2 -23323.728} C_VEL
LIN {X 0,Y 183.732,Z 218.662,A -85,B 0,C 180,E1 -23325.952,E2 -23325.952} C_VEL
LIN {X 0,Y 180.961,Z 210.559,A -85,B 0,C 180,E1 -23326.811,E2 -23326.811} C_VEL
LIN {X 0,Y 173.051,Z 194.201,A -85,B 0,C 180,E1 -23329.123,E2 -23329.123} C_VEL
LIN {X 0,Y 167.529,Z 184.392,A -85,B 0,C 180,E1 -23330.821,E2 -23330.821} C_VEL
LIN {X 0,Y 165.832,Z 181.492,A -85,B 0,C 180,E1 -23331.366,E2 -23331.366} C_VEL
LIN {X 0,Y 164.529,Z 178.822,A -85,B 0,C 180,E1 -23331.819,E2 -23331.819} C_VEL
LIN {X 0,Y 164.368,Z 177.987,A -85,B 0,C 180,E1 -23331.976,E2 -23331.976} C_VEL
LIN {X 0,Y 164.332,Z 177.958,A -85,B 0,C 180,E1 -23336.093,E2 -23336.093} C_VEL
LIN {X 0,Y 164.342,Z 178.013,A -85,B 0,C 180,E1 -23341.211,E2 -23341.211} C_VEL
LIN {X 0,Y 164.277,Z 177.998,A -85,B 0,C 180,E1 -23346.795,E2 -23346.795} C_VEL
LIN {X 0,Y 164.284,Z 178.02,A -85,B 0,C 180,E1 -23349.919,E2 -23349.919} C_VEL
LIN {X 0,Y 164.278,Z 178.012,A -85,B 0,C 180,E1 -23353.343,E2 -23353.343} C_VEL
LIN {X 0,Y 164.258,Z 177.987,A -85,B 0,C 180,E1 -23356.799,E2 -23356.799} C_VEL
LIN {X 0,Y 164.288,Z 178.01,A -85,B 0,C 180,E1 -23360.356,E2 -23360.356} C_VEL
LIN {X 0,Y 164.325,Z 178.012,A -85,B 0,C 180,E1 -23364.353,E2 -23364.353} C_VEL
LIN {X 0,Y 164.367,Z 177.964,A -85,B 0,C 180,E1 -23369.131,E2 -23369.131} C_VEL
LIN {X 0,Y 164.358,Z 177.995,A -85,B 0,C 180,E1 -23374.686,E2 -23374.686} C_VEL
LIN {X 0,Y 164.417,Z 178.001,A -85,B 0,C 180,E1 -23380.119,E2 -23380.119} C_VEL
LIN {X 0,Y 164.471,Z 177.995,A -85,B 0,C 180,E1 -23385.146,E2 -23385.146} C_VEL
LIN {X 0,Y 164.765,Z 177.949,A -85,B 0,C 180,E1 -23390.178,E2 -23390.178} C_VEL
LIN {X 0,Y 164.821,Z 177.947,A -85,B 0,C 180,E1 -23392.652,E2 -23392.652} C_VEL
LIN {X 0,Y 165.277,Z 177.885,A -85,B 0,C 180,E1 -23400.001,E2 -23400.001} C_VEL
LIN {X 0,Y 164.823,Z 177.944,A -85,B 0,C 180,E1 -23407.351,E2 -23407.351} C_VEL
LIN {X 0,Y 164.705,Z 177.968,A -85,B 0,C 180,E1 -23411.059,E2 -23411.059} C_VEL
LIN {X 0,Y 164.434,Z 177.994,A -85,B 0,C 180,E1 -23417.41,E2 -23417.41} C_VEL
LIN {X 0,Y 164.355,Z 178.011,A -85,B 0,C 180,E1 -23422.636,E2 -23422.636} C_VEL
LIN {X 0,Y 164.374,Z 178.009,A -85,B 0,C 180,E1 -23426.118,E2 -23426.118} C_VEL
LIN {X 0,Y 164.361,Z 178.013,A -85,B 0,C 180,E1 -23431.218,E2 -23431.218} C_VEL
LIN {X 0,Y 164.284,Z 178.024,A -85,B 0,C 180,E1 -23436.794,E2 -23436.794} C_VEL
LIN {X 0,Y 164.289,Z 178.024,A -85,B 0,C 180,E1 -23439.918,E2 -23439.918} C_VEL
LIN {X 0,Y 164.274,Z 178.027,A -85,B 0,C 180,E1 -23444.903,E2 -23444.903} C_VEL
LIN {X 0,Y 164.314,Z 178.189,A -85,B 0,C 180,E1 -23446.647,E2 -23446.647} C_VEL
LIN {X 0,Y 164.825,Z 180.198,A -85,B 0,C 180,E1 -23447.804,E2 -23447.804} C_VEL
LIN {X 0,Y 171.319,Z 193.957,A -85,B 0,C 180,E1 -23449.98,E2 -23449.98} C_VEL
LIN {X 0,Y 177.095,Z 208.192,A -85,B 0,C 180,E1 -23451.839,E2 -23451.839} C_VEL
LIN {X 0,Y 180.603,Z 218.566,A -85,B 0,C 180,E1 -23452.974,E2 -23452.974} C_VEL
LIN {X 0,Y 182.819,Z 241.491,A -85,B 0,C 180,E1 -23454.41,E2 -23454.41} C_VEL
LIN {X 0,Y 180.455,Z 289.715,A -85,B 0,C 180,E1 -23456.282,E2 -23456.282} C_VEL
LIN {X 0,Y 178.998,Z 303.51,A -85,B 0,C 180,E1 -23457.241,E2 -23457.241} C_VEL
LIN {X 0,Y 177.236,Z 315.349,A -85,B 0,C 180,E1 -23458.47,E2 -23458.47} C_VEL
LIN {X 0,Y 174.964,Z 327.373,A -85,B 0,C 180,E1 -23460.192,E2 -23460.192} C_VEL
LIN {X 0,Y 172.762,Z 337.607,A -85,B 0,C 180,E1 -23462.106,E2 -23462.106} C_VEL
LIN {X 0,Y 172.073,Z 340.516,A -85,B 0,C 180,E1 -23462.728,E2 -23462.728} C_VEL
LIN {X 0,Y 170.398,Z 345.239,A -85,B 0,C 180,E1 -23463.79,E2 -23463.79} C_VEL
LIN {X 0,Y 165.915,Z 352.47,A -85,B 0,C 180,E1 -23465.531,E2 -23465.531} C_VEL
LIN {X 0,Y 162.164,Z 357.849,A -85,B 0,C 180,E1 -23467.089,E2 -23467.089} C_VEL
LIN {X 0,Y 160.045,Z 361.762,A -85,B 0,C 180,E1 -23468.473,E2 -23468.473} C_VEL
LIN {X 0,Y 159.586,Z 363.024,A -85,B 0,C 180,E1 -23468.983,E2 -23468.983} C_VEL
LIN {X 0,Y 157.671,Z 370.629,A -85,B 0,C 180,E1 -23472.489,E2 -23472.489} C_VEL
LIN {X 0,Y 156.285,Z 376.203,A -85,B 0,C 180,E1 -23475.68,E2 -23475.68} C_VEL
LIN {X 0,Y 155.376,Z 381.653,A -85,B 0,C 180,E1 -23479.576,E2 -23479.576} C_VEL
LIN {X 0,Y 154.905,Z 385.869,A -85,B 0,C 180,E1 -23483.487,E2 -23483.487} C_VEL
LIN {X 0,Y 154.848,Z 388.984,A -85,B 0,C 180,E1 -23487.398,E2 -23487.398} C_VEL
LIN {X 0,Y 154.987,Z 390.517,A -85,B 0,C 180,E1 -23490,E2 -23490} C_VEL
LIN {X 0,Y 154.817,Z 391.662,A -85,B 0,C 180,E1 -23492.894,E2 -23492.894} C_VEL
LIN {X 0,Y 154.961,Z 392.489,A -85,B 0,C 180,E1 -23497.819,E2 -23497.819} C_VEL
LIN {X 0,Y 156.086,Z 391.886,A -85,B 0,C 180,E1 -23503.01,E2 -23503.01} C_VEL
LIN {X 0,Y 158.375,Z 389.683,A -85,B 0,C 180,E1 -23508.097,E2 -23508.097} C_VEL
LIN {X 0,Y 162.049,Z 385.903,A -85,B 0,C 180,E1 -23512.975,E2 -23512.975} C_VEL
LIN {X 0,Y 165.555,Z 381.883,A -85,B 0,C 180,E1 -23516.47,E2 -23516.47} C_VEL
LIN {X 0,Y 170.205,Z 375.765,A -85,B 0,C 180,E1 -23520.386,E2 -23520.386} C_VEL
LIN {X 0,Y 175.012,Z 369.125,A -85,B 0,C 180,E1 -23523.515,E2 -23523.515} C_VEL
LIN {X 0,Y 180.456,Z 360.915,A -85,B 0,C 180,E1 -23526.436,E2 -23526.436} C_VEL
LIN {X 0,Y 185.29,Z 352.553,A -85,B 0,C 180,E1 -23528.744,E2 -23528.744} C_VEL
LIN {X 0,Y 189.352,Z 344.529,A -85,B 0,C 180,E1 -23530.506,E2 -23530.506} C_VEL
LIN {X 0,Y 194.248,Z 333.599,A -85,B 0,C 180,E1 -23532.366,E2 -23532.366} C_VEL
LIN {X 0,Y 198.284,Z 322.925,A -85,B 0,C 180,E1 -23533.722,E2 -23533.722} C_VEL
LIN {X 0,Y 201.956,Z 310.635,A -85,B 0,C 180,E1 -23534.904,E2 -23534.904} C_VEL
LIN {X 0,Y 204.878,Z 297.766,A -85,B 0,C 180,E1 -23535.757,E2 -23535.757} C_VEL
LIN {X 0,Y 206.631,Z 285.098,A -85,B 0,C 180,E1 -23536.338,E2 -23536.338} C_VEL
LIN {X 0,Y 208.842,Z 255.892,A -85,B 0,C 180,E1 -23537.291,E2 -23537.291} C_VEL
LIN {X 0,Y 205.083,Z 246.351,A -85,B 0,C 180,E1 -23539.444,E2 -23539.444} C_VEL
LIN {X 0,Y 200.418,Z 236.367,A -85,B 0,C 180,E1 -23542.297,E2 -23542.297} C_VEL
LIN {X 0,Y 196.723,Z 229.28,A -85,B 0,C 180,E1 -23544.825,E2 -23544.825} C_VEL
LIN {X 0,Y 194.009,Z 224.373,A -85,B 0,C 180,E1 -23546.891,E2 -23546.891} C_VEL
LIN {X 0,Y 191.9,Z 220.74,A -85,B 0,C 180,E1 -23548.644,E2 -23548.644} C_VEL
LIN {X 0,Y 188.837,Z 215.635,A -85,B 0,C 180,E1 -23551.505,E2 -23551.505} C_VEL
LIN {X 0,Y 185.403,Z 210.182,A -85,B 0,C 180,E1 -23555.519,E2 -23555.519} C_VEL
LIN {X 0,Y 183.258,Z 207.45,A -85,B 0,C 180,E1 -23558.633,E2 -23558.633} C_VEL
LIN {X 0,Y 181.483,Z 204.687,A -85,B 0,C 180,E1 -23562.27,E2 -23562.27} C_VEL
LIN {X 0,Y 181.097,Z 203.364,A -85,B 0,C 180,E1 -23563.585,E2 -23563.585} C_VEL
LIN {X 0,Y 179.872,Z 202.682,A -85,B 0,C 180,E1 -23571.007,E2 -23571.007} C_VEL
LIN {X 0,Y 181.65,Z 203.339,A -85,B 0,C 180,E1 -23578.254,E2 -23578.254} C_VEL
LIN {X 0,Y 182.987,Z 206.624,A -85,B 0,C 180,E1 -23581.374,E2 -23581.374} C_VEL
LIN {X 0,Y 185.442,Z 208.947,A -85,B 0,C 180,E1 -23584.89,E2 -23584.89} C_VEL
LIN {X 0,Y 187.667,Z 212.43,A -85,B 0,C 180,E1 -23587.62,E2 -23587.62} C_VEL
LIN {X 0,Y 188.979,Z 214.017,A -85,B 0,C 180,E1 -23588.978,E2 -23588.978} C_VEL
LIN {X 0,Y 191.615,Z 217.788,A -85,B 0,C 180,E1 -23591.413,E2 -23591.413} C_VEL
LIN {X 0,Y 193.282,Z 220.219,A -85,B 0,C 180,E1 -23592.801,E2 -23592.801} C_VEL
LIN {X 0,Y 195.742,Z 223.857,A -85,B 0,C 180,E1 -23594.688,E2 -23594.688} C_VEL
LIN {X 0,Y 199.954,Z 230.231,A -85,B 0,C 180,E1 -23597.567,E2 -23597.567} C_VEL
LIN {X 0,Y 205.242,Z 239.097,A -85,B 0,C 180,E1 -23600.694,E2 -23600.694} C_VEL
LIN {X 0,Y 208.87,Z 246.561,A -85,B 0,C 180,E1 -23602.693,E2 -23602.693} C_VEL
LIN {X 0,Y 209.468,Z 247.968,A -85,B 0,C 180,E1 -23603.017,E2 -23603.017} C_VEL
LIN {X 0,Y 206.838,Z 279.975,A -85,B 0,C 180,E1 -23604.062,E2 -23604.062} C_VEL
LIN {X 0,Y 204.603,Z 293.655,A -85,B 0,C 180,E1 -23604.804,E2 -23604.804} C_VEL
LIN {X 0,Y 201.647,Z 306.372,A -85,B 0,C 180,E1 -23605.889,E2 -23605.889} C_VEL
LIN {X 0,Y 197.752,Z 318.728,A -85,B 0,C 180,E1 -23607.316,E2 -23607.316} C_VEL
LIN {X 0,Y 193.649,Z 329.346,A -85,B 0,C 180,E1 -23608.954,E2 -23608.954} C_VEL
LIN {X 0,Y 188.701,Z 339.879,A -85,B 0,C 180,E1 -23611.062,E2 -23611.062} C_VEL
LIN {X 0,Y 183.465,Z 349.445,A -85,B 0,C 180,E1 -23613.573,E2 -23613.573} C_VEL
LIN {X 0,Y 178.723,Z 357.027,A -85,B 0,C 180,E1 -23616.145,E2 -23616.145} C_VEL
LIN {X 0,Y 174.082,Z 363.595,A -85,B 0,C 180,E1 -23618.999,E2 -23618.999} C_VEL
LIN {X 0,Y 170.06,Z 368.787,A -85,B 0,C 180,E1 -23621.937,E2 -23621.937} C_VEL
LIN {X 0,Y 165.896,Z 373.585,A -85,B 0,C 180,E1 -23625.501,E2 -23625.501} C_VEL
LIN {X 0,Y 162.212,Z 377.352,A -85,B 0,C 180,E1 -23629.467,E2 -23629.467} C_VEL
LIN {X 0,Y 160.207,Z 379.123,A -85,B 0,C 180,E1 -23632.148,E2 -23632.148} C_VEL
LIN {X 0,Y 158.53,Z 380.402,A -85,B 0,C 180,E1 -23634.808,E2 -23634.808} C_VEL
LIN {X 0,Y 156.815,Z 381.358,A -85,B 0,C 180,E1 -23638.375,E2 -23638.375} C_VEL
LIN {X 0,Y 155.286,Z 381.472,A -85,B 0,C 180,E1 -23643.091,E2 -23643.091} C_VEL
LIN {X 0,Y 154.82,Z 380.924,A -85,B 0,C 180,E1 -23645.886,E2 -23645.886} C_VEL
LIN {X 0,Y 154.479,Z 379.917,A -85,B 0,C 180,E1 -23648.657,E2 -23648.657} C_VEL
LIN {X 0,Y 154.53,Z 377.611,A -85,B 0,C 180,E1 -23652.756,E2 -23652.756} C_VEL
LIN {X 0,Y 155.073,Z 374.181,A -85,B 0,C 180,E1 -23656.903,E2 -23656.903} C_VEL
LIN {X 0,Y 156.015,Z 369.741,A -85,B 0,C 180,E1 -23660.867,E2 -23660.867} C_VEL
LIN {X 0,Y 157.367,Z 363.911,A -85,B 0,C 180,E1 -23664.876,E2 -23664.876} C_VEL
LIN {X 0,Y 159.217,Z 356.715,A -85,B 0,C 180,E1 -23668.736,E2 -23668.736} C_VEL
LIN {X 0,Y 161.655,Z 347.67,A -85,B 0,C 180,E1 -23672.492,E2 -23672.492} C_VEL
LIN {X 0,Y 164.113,Z 338.388,A -85,B 0,C 180,E1 -23675.53,E2 -23675.53} C_VEL
LIN {X 0,Y 166.646,Z 328.087,A -85,B 0,C 180,E1 -23678.183,E2 -23678.183} C_VEL
LIN {X 0,Y 169.186,Z 316.592,A -85,B 0,C 180,E1 -23680.472,E2 -23680.472} C_VEL
LIN {X 0,Y 171.258,Z 304.758,A -85,B 0,C 180,E1 -23682.292,E2 -23682.292} C_VEL
LIN {X 0,Y 173.119,Z 291.728,A -85,B 0,C 180,E1 -23683.724,E2 -23683.724} C_VEL
LIN {X 0,Y 174.351,Z 278.987,A -85,B 0,C 180,E1 -23684.67,E2 -23684.67} C_VEL
LIN {X 0,Y 176.245,Z 244.206,A -85,B 0,C 180,E1 -23686.08,E2 -23686.08} C_VEL
LIN {X 0,Y 177.433,Z 219.999,A -85,B 0,C 180,E1 -23687.011,E2 -23687.011} C_VEL
LIN {X 0,Y 174.884,Z 212.828,A -85,B 0,C 180,E1 -23687.839,E2 -23687.839} C_VEL
LIN {X 0,Y 166.958,Z 196.544,A -85,B 0,C 180,E1 -23690.313,E2 -23690.313} C_VEL
LIN {X 0,Y 161.22,Z 186.34,A -85,B 0,C 180,E1 -23692.216,E2 -23692.216} C_VEL
LIN {X 0,Y 158.978,Z 182.628,A -85,B 0,C 180,E1 -23692.984,E2 -23692.984} C_VEL
LIN {X 0,Y 157.57,Z 180.239,A -85,B 0,C 180,E1 -23693.485,E2 -23693.485} C_VEL
LIN {X 0,Y 157.261,Z 178.843,A -85,B 0,C 180,E1 -23693.717,E2 -23693.717} C_VEL
LIN {X 0,Y 157.263,Z 178.839,A -85,B 0,C 180,E1 -23696.65,E2 -23696.65} C_VEL
LIN {X 0,Y 157.258,Z 178.897,A -85,B 0,C 180,E1 -23702.432,E2 -23702.432} C_VEL
LIN {X 0,Y 157.256,Z 178.871,A -85,B 0,C 180,E1 -23706.446,E2 -23706.446} C_VEL
LIN {X 0,Y 157.188,Z 178.903,A -85,B 0,C 180,E1 -23712.119,E2 -23712.119} C_VEL
LIN {X 0,Y 157.188,Z 178.87,A -85,B 0,C 180,E1 -23717.884,E2 -23717.884} C_VEL
LIN {X 0,Y 157.258,Z 178.894,A -85,B 0,C 180,E1 -23723.557,E2 -23723.557} C_VEL
LIN {X 0,Y 157.28,Z 178.855,A -85,B 0,C 180,E1 -23728.106,E2 -23728.106} C_VEL
LIN {X 0,Y 157.267,Z 178.864,A -85,B 0,C 180,E1 -23733.458,E2 -23733.458} C_VEL
LIN {X 0,Y 157.36,Z 178.883,A -85,B 0,C 180,E1 -23739.704,E2 -23739.704} C_VEL
LIN {X 0,Y 157.406,Z 178.871,A -85,B 0,C 180,E1 -23744.462,E2 -23744.462} C_VEL
LIN {X 0,Y 157.688,Z 178.833,A -85,B 0,C 180,E1 -23749.732,E2 -23749.732} C_VEL
LIN {X 0,Y 157.759,Z 178.823,A -85,B 0,C 180,E1 -23752.321,E2 -23752.321} C_VEL
LIN {X 0,Y 158.239,Z 178.762,A -85,B 0,C 180,E1 -23760.001,E2 -23760.001} C_VEL
LIN {X 0,Y 157.761,Z 178.821,A -85,B 0,C 180,E1 -23767.682,E2 -23767.682} C_VEL
LIN {X 0,Y 157.634,Z 178.849,A -85,B 0,C 180,E1 -23771.225,E2 -23771.225} C_VEL
LIN {X 0,Y 157.413,Z 178.865,A -85,B 0,C 180,E1 -23775.54,E2 -23775.54} C_VEL
LIN {X 0,Y 157.314,Z 178.889,A -85,B 0,C 180,E1 -23780.942,E2 -23780.942} C_VEL
LIN {X 0,Y 157.314,Z 178.889,A -85,B 0,C 180,E1 -23786.682,E2 -23786.682} C_VEL
LIN {X 0,Y 157.272,Z 178.895,A -85,B 0,C 180,E1 -23792.43,E2 -23792.43} C_VEL
LIN {X 0,Y 157.262,Z 178.897,A -85,B 0,C 180,E1 -23796.445,E2 -23796.445} C_VEL
LIN {X 0,Y 157.193,Z 178.91,A -85,B 0,C 180,E1 -23802.118,E2 -23802.118} C_VEL
LIN {X 0,Y 157.251,Z 178.981,A -85,B 0,C 180,E1 -23805.458,E2 -23805.458} C_VEL
LIN {X 0,Y 157.409,Z 179.812,A -85,B 0,C 180,E1 -23805.932,E2 -23805.932} C_VEL
LIN {X 0,Y 164.521,Z 194.421,A -85,B 0,C 180,E1 -23808.497,E2 -23808.497} C_VEL
LIN {X 0,Y 169.769,Z 206.879,A -85,B 0,C 180,E1 -23810.309,E2 -23810.309} C_VEL
LIN {X 0,Y 174.569,Z 220.706,A -85,B 0,C 180,E1 -23811.961,E2 -23811.961} C_VEL
LIN {X 0,Y 176.59,Z 241.802,A -85,B 0,C 180,E1 -23813.346,E2 -23813.346} C_VEL
LIN {X 0,Y 174.138,Z 289.52,A -85,B 0,C 180,E1 -23815.25,E2 -23815.25} C_VEL
LIN {X 0,Y 172.633,Z 303.169,A -85,B 0,C 180,E1 -23816.223,E2 -23816.223} C_VEL
LIN {X 0,Y 170.807,Z 315.034,A -85,B 0,C 180,E1 -23817.488,E2 -23817.488} C_VEL
LIN {X 0,Y 168.818,Z 325.463,A -85,B 0,C 180,E1 -23818.99,E2 -23818.99} C_VEL
LIN {X 0,Y 166.137,Z 337.317,A -85,B 0,C 180,E1 -23821.236,E2 -23821.236} C_VEL
LIN {X 0,Y 163.767,Z 346.871,A -85,B 0,C 180,E1 -23823.561,E2 -23823.561} C_VEL
LIN {X 0,Y 161.601,Z 355.134,A -85,B 0,C 180,E1 -23826.052,E2 -23826.052} C_VEL
LIN {X 0,Y 159.586,Z 363.024,A -85,B 0,C 180,E1 -23828.983,E2 -23828.983} C_VEL
LIN {X 0,Y 157.877,Z 366.721,A -85,B 0,C 180,E1 -23830.534,E2 -23830.534} C_VEL
LIN {X 0,Y 153.622,Z 372.202,A -85,B 0,C 180,E1 -23833.147,E2 -23833.147} C_VEL
LIN {X 0,Y 149.694,Z 377.026,A -85,B 0,C 180,E1 -23836.067,E2 -23836.067} C_VEL
LIN {X 0,Y 148.541,Z 379.685,A -85,B 0,C 180,E1 -23838.048,E2 -23838.048} C_VEL
LIN {X 0,Y 147.972,Z 383.988,A -85,B 0,C 180,E1 -23841.808,E2 -23841.808} C_VEL
LIN {X 0,Y 147.73,Z 387.549,A -85,B 0,C 180,E1 -23845.907,E2 -23845.907} C_VEL
LIN {X 0,Y 147.894,Z 390.067,A -85,B 0,C 180,E1 -23850,E2 -23850} C_VEL
LIN {X 0,Y 147.744,Z 391.203,A -85,B 0,C 180,E1 -23852.726,E2 -23852.726} C_VEL
LIN {X 0,Y 147.929,Z 392.208,A -85,B 0,C 180,E1 -23858.194,E2 -23858.194} C_VEL
LIN {X 0,Y 149.141,Z 391.697,A -85,B 0,C 180,E1 -23863.628,E2 -23863.628} C_VEL
LIN {X 0,Y 150.195,Z 390.861,A -85,B 0,C 180,E1 -23866.305,E2 -23866.305} C_VEL
LIN {X 0,Y 153.457,Z 387.972,A -85,B 0,C 180,E1 -23871.492,E2 -23871.492} C_VEL
LIN {X 0,Y 156.682,Z 384.72,A -85,B 0,C 180,E1 -23875.221,E2 -23875.221} C_VEL
LIN {X 0,Y 160.591,Z 380.279,A -85,B 0,C 180,E1 -23878.921,E2 -23878.921} C_VEL
LIN {X 0,Y 165.743,Z 374.014,A -85,B 0,C 180,E1 -23882.727,E2 -23882.727} C_VEL
LIN {X 0,Y 170.988,Z 367.047,A -85,B 0,C 180,E1 -23885.853,E2 -23885.853} C_VEL
LIN {X 0,Y 176.727,Z 358.374,A -85,B 0,C 180,E1 -23888.78,E2 -23888.78} C_VEL
LIN {X 0,Y 181.844,Z 349.542,A -85,B 0,C 180,E1 -23891.073,E2 -23891.073} C_VEL
LIN {X 0,Y 187.41,Z 338.672,A -85,B 0,C 180,E1 -23893.187,E2 -23893.187} C_VEL
LIN {X 0,Y 192.049,Z 327.723,A -85,B 0,C 180,E1 -23894.785,E2 -23894.785} C_VEL
LIN {X 0,Y 196.273,Z 315.512,A -85,B 0,C 180,E1 -23896.105,E2 -23896.105} C_VEL
LIN {X 0,Y 199.372,Z 304.019,A -85,B 0,C 180,E1 -23897.004,E2 -23897.004} C_VEL
LIN {X 0,Y 201.76,Z 291.39,A -85,B 0,C 180,E1 -23897.704,E2 -23897.704} C_VEL
LIN {X 0,Y 203.451,Z 274.428,A -85,B 0,C 180,E1 -23898.312,E2 -23898.312} C_VEL
LIN {X 0,Y 204.617,Z 258.523,A -85,B 0,C 180,E1 -23898.849,E2 -23898.849} C_VEL
LIN {X 0,Y 201.106,Z 249.575,A -85,B 0,C 180,E1 -23901.019,E2 -23901.019} C_VEL
LIN {X 0,Y 197.064,Z 240.637,A -85,B 0,C 180,E1 -23903.717,E2 -23903.717} C_VEL
LIN {X 0,Y 192.64,Z 231.836,A -85,B 0,C 180,E1 -23907.097,E2 -23907.097} C_VEL
LIN {X 0,Y 189.661,Z 226.544,A -85,B 0,C 180,E1 -23909.684,E2 -23909.684} C_VEL
LIN {X 0,Y 186.967,Z 221.854,A -85,B 0,C 180,E1 -23912.402,E2 -23912.402} C_VEL
LIN {X 0,Y 183.93,Z 216.801,A -85,B 0,C 180,E1 -23916.196,E2 -23916.196} C_VEL
LIN {X 0,Y 182.053,Z 214.304,A -85,B 0,C 180,E1 -23919.077,E2 -23919.077} C_VEL
LIN {X 0,Y 180.321,Z 211.327,A -85,B 0,C 180,E1 -23922.962,E2 -23922.962} C_VEL
LIN {X 0,Y 180,Z 210.303,A -85,B 0,C 180,E1 -23924.137,E2 -23924.137} C_VEL
LIN {X 0,Y 178.968,Z 209.726,A -85,B 0,C 180,E1 -23930.961,E2 -23930.961} C_VEL
LIN {X 0,Y 180.576,Z 210.38,A -85,B 0,C 180,E1 -23937.887,E2 -23937.887} C_VEL
LIN {X 0,Y 181.813,Z 213.5,A -85,B 0,C 180,E1 -23940.959,E2 -23940.959} C_VEL
LIN {X 0,Y 184.083,Z 215.809,A -85,B 0,C 180,E1 -23944.378,E2 -23944.378} C_VEL
LIN {X 0,Y 186.52,Z 219.535,A -85,B 0,C 180,E1 -23947.441,E2 -23947.441} C_VEL
LIN {X 0,Y 187.402,Z 220.809,A -85,B 0,C 180,E1 -23948.405,E2 -23948.405} C_VEL
LIN {X 0,Y 190.763,Z 225.691,A -85,B 0,C 180,E1 -23951.587,E2 -23951.587} C_VEL
LIN {X 0,Y 193.734,Z 230.332,A -85,B 0,C 180,E1 -23954.015,E2 -23954.015} C_VEL
LIN {X 0,Y 197.37,Z 235.958,A -85,B 0,C 180,E1 -23956.626,E2 -23956.626} C_VEL
LIN {X 0,Y 202.503,Z 244.956,A -85,B 0,C 180,E1 -23959.86,E2 -23959.86} C_VEL
LIN {X 0,Y 205.263,Z 250.968,A -85,B 0,C 180,E1 -23961.484,E2 -23961.484} C_VEL
LIN {X 0,Y 202.779,Z 280.063,A -85,B 0,C 180,E1 -23962.439,E2 -23962.439} C_VEL
LIN {X 0,Y 200.571,Z 293.269,A -85,B 0,C 180,E1 -23963.142,E2 -23963.142} C_VEL
LIN {X 0,Y 197.779,Z 305.129,A -85,B 0,C 180,E1 -23964.106,E2 -23964.106} C_VEL
LIN {X 0,Y 194.4,Z 316.173,A -85,B 0,C 180,E1 -23965.337,E2 -23965.337} C_VEL
LIN {X 0,Y 190.339,Z 326.592,A -85,B 0,C 180,E1 -23966.811,E2 -23966.811} C_VEL
LIN {X 0,Y 185.455,Z 337.193,A -85,B 0,C 180,E1 -23968.796,E2 -23968.796} C_VEL
LIN {X 0,Y 180.417,Z 346.43,A -85,B 0,C 180,E1 -23971.019,E2 -23971.019} C_VEL
LIN {X 0,Y 175.377,Z 354.485,A -85,B 0,C 180,E1 -23973.525,E2 -23973.525} C_VEL
LIN {X 0,Y 170.273,Z 361.632,A -85,B 0,C 180,E1 -23976.404,E2 -23976.404} C_VEL
LIN {X 0,Y 164.962,Z 368.196,A -85,B 0,C 180,E1 -23979.927,E2 -23979.927} C_VEL
LIN {X 0,Y 160.331,Z 373.315,A -85,B 0,C 180,E1 -23983.675,E2 -23983.675} C_VEL
LIN {X 0,Y 156.379,Z 377.141,A -85,B 0,C 180,E1 -23987.614,E2 -23987.614} C_VEL
LIN {X 0,Y 153.679,Z 379.407,A -85,B 0,C 180,E1 -23991.024,E2 -23991.024} C_VEL
LIN {X 0,Y 150.722,Z 381.346,A -85,B 0,C 180,E1 -23995.976,E2 -23995.976} C_VEL
LIN {X 0,Y 149.447,Z 381.798,A -85,B 0,C 180,E1 -23998.849,E2 -23998.849} C_VEL
LIN {X 0,Y 148.487,Z 381.787,A -85,B 0,C 180,E1 -24001.751,E2 -24001.751} C_VEL
LIN {X 0,Y 147.893,Z 381.349,A -85,B 0,C 180,E1 -24004.68,E2 -24004.68} C_VEL
LIN {X 0,Y 147.472,Z 380.453,A -85,B 0,C 180,E1 -24007.589,E2 -24007.589} C_VEL
LIN {X 0,Y 147.425,Z 377.932,A -85,B 0,C 180,E1 -24012.441,E2 -24012.441} C_VEL
LIN {X 0,Y 148.107,Z 373.707,A -85,B 0,C 180,E1 -24017.671,E2 -24017.671} C_VEL
LIN {X 0,Y 149.13,Z 368.974,A -85,B 0,C 180,E1 -24021.873,E2 -24021.873} C_VEL
LIN {X 0,Y 150.654,Z 362.94,A -85,B 0,C 180,E1 -24025.988,E2 -24025.988} C_VEL
LIN {X 0,Y 152.686,Z 355.409,A -85,B 0,C 180,E1 -24030,E2 -24030} C_VEL
LIN {X 0,Y 155.16,Z 346.722,A -85,B 0,C 180,E1 -24033.634,E2 -24033.634} C_VEL
LIN {X 0,Y 157.79,Z 337.326,A -85,B 0,C 180,E1 -24036.715,E2 -24036.715} C_VEL
LIN {X 0,Y 160.43,Z 326.695,A -85,B 0,C 180,E1 -24039.456,E2 -24039.456} C_VEL
LIN {X 0,Y 163.125,Z 314.828,A -85,B 0,C 180,E1 -24041.809,E2 -24041.809} C_VEL
LIN {X 0,Y 165.135,Z 303.384,A -85,B 0,C 180,E1 -24043.538,E2 -24043.538} C_VEL
LIN {X 0,Y 166.991,Z 290.019,A -85,B 0,C 180,E1 -24044.987,E2 -24044.987} C_VEL
LIN {X 0,Y 168.312,Z 276.647,A -85,B 0,C 180,E1 -24045.919,E2 -24045.919} C_VEL
LIN {X 0,Y 171.351,Z 222.1,A -85,B 0,C 180,E1 -24048.079,E2 -24048.079} C_VEL
LIN {X 0,Y 169.558,Z 216.74,A -85,B 0,C 180,E1 -24048.713,E2 -24048.713} C_VEL
LIN {X 0,Y 161.836,Z 200.557,A -85,B 0,C 180,E1 -24051.285,E2 -24051.285} C_VEL
LIN {X 0,Y 155.803,Z 189.821,A -85,B 0,C 180,E1 -24053.403,E2 -24053.403} C_VEL
LIN {X 0,Y 152.088,Z 183.732,A -85,B 0,C 180,E1 -24054.785,E2 -24054.785} C_VEL
LIN {X 0,Y 150.564,Z 181.264,A -85,B 0,C 180,E1 -24055.378,E2 -24055.378} C_VEL
LIN {X 0,Y 150.176,Z 179.715,A -85,B 0,C 180,E1 -24055.653,E2 -24055.653} C_VEL
LIN {X 0,Y 150.178,Z 179.776,A -85,B 0,C 180,E1 -24060.983,E2 -24060.983} C_VEL
LIN {X 0,Y 150.18,Z 179.763,A -85,B 0,C 180,E1 -24064.165,E2 -24064.165} C_VEL
LIN {X 0,Y 150.167,Z 179.757,A -85,B 0,C 180,E1 -24067.476,E2 -24067.476} C_VEL
LIN {X 0,Y 150.131,Z 179.783,A -85,B 0,C 180,E1 -24071.499,E2 -24071.499} C_VEL
LIN {X 0,Y 150.124,Z 179.749,A -85,B 0,C 180,E1 -24075.397,E2 -24075.397} C_VEL
LIN {X 0,Y 150.135,Z 179.758,A -85,B 0,C 180,E1 -24079.055,E2 -24079.055} C_VEL
LIN {X 0,Y 150.175,Z 179.777,A -85,B 0,C 180,E1 -24082.711,E2 -24082.711} C_VEL
LIN {X 0,Y 150.205,Z 179.742,A -85,B 0,C 180,E1 -24087.376,E2 -24087.376} C_VEL
LIN {X 0,Y 150.184,Z 179.736,A -85,B 0,C 180,E1 -24092.765,E2 -24092.765} C_VEL
LIN {X 0,Y 150.283,Z 179.764,A -85,B 0,C 180,E1 -24099.28,E2 -24099.28} C_VEL
LIN {X 0,Y 150.311,Z 179.751,A -85,B 0,C 180,E1 -24103.709,E2 -24103.709} C_VEL
LIN {X 0,Y 150.608,Z 179.719,A -85,B 0,C 180,E1 -24109.244,E2 -24109.244} C_VEL
LIN {X 0,Y 150.682,Z 179.702,A -85,B 0,C 180,E1 -24111.958,E2 -24111.958} C_VEL
LIN {X 0,Y 151.199,Z 179.638,A -85,B 0,C 180,E1 -24120.001,E2 -24120.001} C_VEL
LIN {X 0,Y 150.684,Z 179.702,A -85,B 0,C 180,E1 -24128.045,E2 -24128.045} C_VEL
LIN {X 0,Y 150.577,Z 179.729,A -85,B 0,C 180,E1 -24131.43,E2 -24131.43} C_VEL
LIN {X 0,Y 150.318,Z 179.747,A -85,B 0,C 180,E1 -24136.293,E2 -24136.293} C_VEL
LIN {X 0,Y 150.288,Z 179.765,A -85,B 0,C 180,E1 -24140.725,E2 -24140.725} C_VEL
LIN {X 0,Y 150.243,Z 179.771,A -85,B 0,C 180,E1 -24147.278,E2 -24147.278} C_VEL
LIN {X 0,Y 150.212,Z 179.774,A -85,B 0,C 180,E1 -24152.629,E2 -24152.629} C_VEL
LIN {X 0,Y 150.173,Z 179.781,A -85,B 0,C 180,E1 -24157.475,E2 -24157.475} C_VEL
LIN {X 0,Y 150.144,Z 179.788,A -85,B 0,C 180,E1 -24162.915,E2 -24162.915} C_VEL
LIN {X 0,Y 150.16,Z 179.785,A -85,B 0,C 180,E1 -24163.851,E2 -24163.851} C_VEL
LIN {X 0,Y 151.377,Z 182.937,A -85,B 0,C 180,E1 -24164.446,E2 -24164.446} C_VEL
LIN {X 0,Y 152.839,Z 184.953,A -85,B 0,C 180,E1 -24164.985,E2 -24164.985} C_VEL
LIN {X 0,Y 158.726,Z 196.86,A -85,B 0,C 180,E1 -24167.23,E2 -24167.23} C_VEL
LIN {X 0,Y 164.056,Z 209.71,A -85,B 0,C 180,E1 -24169.207,E2 -24169.207} C_VEL
LIN {X 0,Y 168.515,Z 222.379,A -85,B 0,C 180,E1 -24170.835,E2 -24170.835} C_VEL
LIN {X 0,Y 170.369,Z 242.632,A -85,B 0,C 180,E1 -24172.224,E2 -24172.224} C_VEL
LIN {X 0,Y 167.886,Z 288.947,A -85,B 0,C 180,E1 -24174.121,E2 -24174.121} C_VEL
LIN {X 0,Y 166.328,Z 302.753,A -85,B 0,C 180,E1 -24175.127,E2 -24175.127} C_VEL
LIN {X 0,Y 164.429,Z 314.66,A -85,B 0,C 180,E1 -24176.428,E2 -24176.428} C_VEL
LIN {X 0,Y 162.362,Z 325.117,A -85,B 0,C 180,E1 -24177.977,E2 -24177.977} C_VEL
LIN {X 0,Y 159.562,Z 336.99,A -85,B 0,C 180,E1 -24180.296,E2 -24180.296} C_VEL
LIN {X 0,Y 157.08,Z 346.555,A -85,B 0,C 180,E1 -24182.703,E2 -24182.703} C_VEL
LIN {X 0,Y 154.885,Z 354.711,A -85,B 0,C 180,E1 -24185.253,E2 -24185.253} C_VEL
LIN {X 0,Y 152.68,Z 362.84,A -85,B 0,C 180,E1 -24188.392,E2 -24188.392} C_VEL
LIN {X 0,Y 150.519,Z 370.959,A -85,B 0,C 180,E1 -24192.332,E2 -24192.332} C_VEL
LIN {X 0,Y 148.966,Z 377.43,A -85,B 0,C 180,E1 -24196.355,E2 -24196.355} C_VEL
LIN {X 0,Y 148.541,Z 379.685,A -85,B 0,C 180,E1 -24198.048,E2 -24198.048} C_VEL
LIN {X 0,Y 147.498,Z 382.167,A -85,B 0,C 180,E1 -24200.098,E2 -24200.098} C_VEL
LIN {X 0,Y 145.641,Z 384.262,A -85,B 0,C 180,E1 -24202.152,E2 -24202.152} C_VEL
LIN {X 0,Y 141.726,Z 387.631,A -85,B 0,C 180,E1 -24206.467,E2 -24206.467} C_VEL
LIN {X 0,Y 140.789,Z 389.01,A -85,B 0,C 180,E1 -24208.788,E2 -24208.788} C_VEL
LIN {X 0,Y 140.775,Z 389.383,A -85,B 0,C 180,E1 -24209.576,E2 -24209.576} C_VEL
LIN {X 0,Y 140.656,Z 390.799,A -85,B 0,C 180,E1 -24212.864,E2 -24212.864} C_VEL
LIN {X 0,Y 140.63,Z 391.573,A -85,B 0,C 180,E1 -24215.736,E2 -24215.736} C_VEL
LIN {X 0,Y 141.397,Z 391.898,A -85,B 0,C 180,E1 -24221.467,E2 -24221.467} C_VEL
LIN {X 0,Y 143.36,Z 390.726,A -85,B 0,C 180,E1 -24227.106,E2 -24227.106} C_VEL
LIN {X 0,Y 144.932,Z 389.541,A -85,B 0,C 180,E1 -24229.842,E2 -24229.842} C_VEL
LIN {X 0,Y 149.039,Z 385.95,A -85,B 0,C 180,E1 -24235.112,E2 -24235.112} C_VEL
LIN {X 0,Y 153.398,Z 381.621,A -85,B 0,C 180,E1 -24239.281,E2 -24239.281} C_VEL
LIN {X 0,Y 157.308,Z 377.222,A -85,B 0,C 180,E1 -24242.42,E2 -24242.42} C_VEL
LIN {X 0,Y 162.483,Z 371.088,A -85,B 0,C 180,E1 -24245.727,E2 -24245.727} C_VEL
LIN {X 0,Y 168.294,Z 363.496,A -85,B 0,C 180,E1 -24248.785,E2 -24248.785} C_VEL
LIN {X 0,Y 173.441,Z 355.774,A -85,B 0,C 180,E1 -24251.183,E2 -24251.183} C_VEL
LIN {X 0,Y 178.853,Z 346.401,A -85,B 0,C 180,E1 -24253.445,E2 -24253.445} C_VEL
LIN {X 0,Y 184.701,Z 334.745,A -85,B 0,C 180,E1 -24255.516,E2 -24255.516} C_VEL
LIN {X 0,Y 188.991,Z 324.523,A -85,B 0,C 180,E1 -24256.869,E2 -24256.869} C_VEL
LIN {X 0,Y 193.044,Z 312.402,A -85,B 0,C 180,E1 -24258.077,E2 -24258.077} C_VEL
LIN {X 0,Y 196.521,Z 298.589,A -85,B 0,C 180,E1 -24259.024,E2 -24259.024} C_VEL
LIN {X 0,Y 198.536,Z 285.91,A -85,B 0,C 180,E1 -24259.627,E2 -24259.627} C_VEL
LIN {X 0,Y 200.627,Z 261.469,A -85,B 0,C 180,E1 -24260.414,E2 -24260.414} C_VEL
LIN {X 0,Y 197.21,Z 252.612,A -85,B 0,C 180,E1 -24262.71,E2 -24262.71} C_VEL
LIN {X 0,Y 193.594,Z 244.543,A -85,B 0,C 180,E1 -24265.381,E2 -24265.381} C_VEL
LIN {X 0,Y 190.14,Z 237.39,A -85,B 0,C 180,E1 -24268.255,E2 -24268.255} C_VEL
LIN {X 0,Y 187.612,Z 232.672,A -85,B 0,C 180,E1 -24270.613,E2 -24270.613} C_VEL
LIN {X 0,Y 185.231,Z 228.218,A -85,B 0,C 180,E1 -24273.219,E2 -24273.219} C_VEL
LIN {X 0,Y 182.523,Z 223.475,A -85,B 0,C 180,E1 -24276.826,E2 -24276.826} C_VEL
LIN {X 0,Y 180.859,Z 221.159,A -85,B 0,C 180,E1 -24279.528,E2 -24279.528} C_VEL
LIN {X 0,Y 179.214,Z 218.109,A -85,B 0,C 180,E1 -24283.542,E2 -24283.542} C_VEL
LIN {X 0,Y 178.982,Z 217.309,A -85,B 0,C 180,E1 -24284.476,E2 -24284.476} C_VEL
LIN {X 0,Y 178.067,Z 216.753,A -85,B 0,C 180,E1 -24290.915,E2 -24290.915} C_VEL
LIN {X 0,Y 179.52,Z 217.423,A -85,B 0,C 180,E1 -24297.543,E2 -24297.543} C_VEL
LIN {X 0,Y 180.742,Z 220.482,A -85,B 0,C 180,E1 -24300.709,E2 -24300.709} C_VEL
LIN {X 0,Y 182.761,Z 222.684,A -85,B 0,C 180,E1 -24303.887,E2 -24303.887} C_VEL
LIN {X 0,Y 185.279,Z 226.502,A -85,B 0,C 180,E1 -24307.149,E2 -24307.149} C_VEL
LIN {X 0,Y 188.965,Z 232.265,A -85,B 0,C 180,E1 -24310.937,E2 -24310.937} C_VEL
LIN {X 0,Y 191.564,Z 236.475,A -85,B 0,C 180,E1 -24313.172,E2 -24313.172} C_VEL
LIN {X 0,Y 195.059,Z 242.147,A -85,B 0,C 180,E1 -24315.825,E2 -24315.825} C_VEL
LIN {X 0,Y 199.488,Z 250.256,A -85,B 0,C 180,E1 -24318.807,E2 -24318.807} C_VEL
LIN {X 0,Y 201.215,Z 254.025,A -85,B 0,C 180,E1 -24319.893,E2 -24319.893} C_VEL
LIN {X 0,Y 198.844,Z 280.461,A -85,B 0,C 180,E1 -24320.764,E2 -24320.764} C_VEL
LIN {X 0,Y 196.6,Z 293.443,A -85,B 0,C 180,E1 -24321.45,E2 -24321.45} C_VEL
LIN {X 0,Y 193.476,Z 306.119,A -85,B 0,C 180,E1 -24322.479,E2 -24322.479} C_VEL
LIN {X 0,Y 189.465,Z 318.28,A -85,B 0,C 180,E1 -24323.868,E2 -24323.868} C_VEL
LIN {X 0,Y 184.916,Z 329.191,A -85,B 0,C 180,E1 -24325.491,E2 -24325.491} C_VEL
LIN {X 0,Y 180.294,Z 338.571,A -85,B 0,C 180,E1 -24327.318,E2 -24327.318} C_VEL
LIN {X 0,Y 175.437,Z 346.99,A -85,B 0,C 180,E1 -24329.39,E2 -24329.39} C_VEL
LIN {X 0,Y 169.959,Z 355.289,A -85,B 0,C 180,E1 -24332.033,E2 -24332.033} C_VEL
LIN {X 0,Y 163.845,Z 363.269,A -85,B 0,C 180,E1 -24335.414,E2 -24335.414} C_VEL
LIN {X 0,Y 158.222,Z 369.728,A -85,B 0,C 180,E1 -24339.151,E2 -24339.151} C_VEL
LIN {X 0,Y 152.798,Z 375.11,A -85,B 0,C 180,E1 -24343.622,E2 -24343.622} C_VEL
LIN {X 0,Y 148.297,Z 378.931,A -85,B 0,C 180,E1 -24348.434,E2 -24348.434} C_VEL
LIN {X 0,Y 146.167,Z 380.422,A -85,B 0,C 180,E1 -24351.313,E2 -24351.313} C_VEL
LIN {X 0,Y 143.302,Z 381.889,A -85,B 0,C 180,E1 -24356.481,E2 -24356.481} C_VEL
LIN {X 0,Y 141.79,Z 382.102,A -85,B 0,C 180,E1 -24360.287,E2 -24360.287} C_VEL
LIN {X 0,Y 140.897,Z 381.644,A -85,B 0,C 180,E1 -24363.873,E2 -24363.873} C_VEL
LIN {X 0,Y 140.496,Z 380.958,A -85,B 0,C 180,E1 -24366.411,E2 -24366.411} C_VEL
LIN {X 0,Y 140.275,Z 379.704,A -85,B 0,C 180,E1 -24369.47,E2 -24369.47} C_VEL
LIN {X 0,Y 140.445,Z 376.971,A -85,B 0,C 180,E1 -24374.025,E2 -24374.025} C_VEL
LIN {X 0,Y 141.164,Z 373.156,A -85,B 0,C 180,E1 -24378.514,E2 -24378.514} C_VEL
LIN {X 0,Y 142.387,Z 367.937,A -85,B 0,C 180,E1 -24383.096,E2 -24383.096} C_VEL
LIN {X 0,Y 144.009,Z 361.9,A -85,B 0,C 180,E1 -24387.203,E2 -24387.203} C_VEL
LIN {X 0,Y 146.248,Z 354.094,A -85,B 0,C 180,E1 -24391.377,E2 -24391.377} C_VEL
LIN {X 0,Y 148.689,Z 345.9,A -85,B 0,C 180,E1 -24394.804,E2 -24394.804} C_VEL
LIN {X 0,Y 151.48,Z 336.218,A -85,B 0,C 180,E1 -24398.001,E2 -24398.001} C_VEL
LIN {X 0,Y 154.339,Z 325.288,A -85,B 0,C 180,E1 -24400.827,E2 -24400.827} C_VEL
LIN {X 0,Y 156.795,Z 314.657,A -85,B 0,C 180,E1 -24402.951,E2 -24402.951} C_VEL
LIN {X 0,Y 158.901,Z 303.065,A -85,B 0,C 180,E1 -24404.734,E2 -24404.734} C_VEL
LIN {X 0,Y 160.775,Z 290.048,A -85,B 0,C 180,E1 -24406.174,E2 -24406.174} C_VEL
LIN {X 0,Y 162.038,Z 277.761,A -85,B 0,C 180,E1 -24407.069,E2 -24407.069} C_VEL
LIN {X 0,Y 165.157,Z 223.07,A -85,B 0,C 180,E1 -24409.323,E2 -24409.323} C_VEL
LIN {X 0,Y 160.312,Z 211.928,A -85,B 0,C 180,E1 -24411.028,E2 -24411.028} C_VEL
LIN {X 0,Y 153.56,Z 198.623,A -85,B 0,C 180,E1 -24413.493,E2 -24413.493} C_VEL
LIN {X 0,Y 147.458,Z 188.44,A -85,B 0,C 180,E1 -24415.86,E2 -24415.86} C_VEL
LIN {X 0,Y 145.097,Z 184.669,A -85,B 0,C 180,E1 -24416.841,E2 -24416.841} C_VEL
LIN {X 0,Y 143.535,Z 182.24,A -85,B 0,C 180,E1 -24417.51,E2 -24417.51} C_VEL
LIN {X 0,Y 143.114,Z 180.608,A -85,B 0,C 180,E1 -24417.796,E2 -24417.796} C_VEL
LIN {X 0,Y 143.131,Z 180.65,A -85,B 0,C 180,E1 -24423.415,E2 -24423.415} C_VEL
LIN {X 0,Y 143.05,Z 180.663,A -85,B 0,C 180,E1 -24429.695,E2 -24429.695} C_VEL
LIN {X 0,Y 143.031,Z 180.652,A -85,B 0,C 180,E1 -24433.466,E2 -24433.466} C_VEL
LIN {X 0,Y 143.035,Z 180.627,A -85,B 0,C 180,E1 -24437.48,E2 -24437.48} C_VEL
LIN {X 0,Y 143.071,Z 180.66,A -85,B 0,C 180,E1 -24441.811,E2 -24441.811} C_VEL
LIN {X 0,Y 143.172,Z 180.617,A -85,B 0,C 180,E1 -24447.321,E2 -24447.321} C_VEL
LIN {X 0,Y 143.106,Z 180.627,A -85,B 0,C 180,E1 -24453.771,E2 -24453.771} C_VEL
LIN {X 0,Y 143.246,Z 180.639,A -85,B 0,C 180,E1 -24459.915,E2 -24459.915} C_VEL
LIN {X 0,Y 143.305,Z 180.633,A -85,B 0,C 180,E1 -24465.807,E2 -24465.807} C_VEL
LIN {X 0,Y 143.534,Z 180.602,A -85,B 0,C 180,E1 -24468.707,E2 -24468.707} C_VEL
LIN {X 0,Y 143.608,Z 180.581,A -85,B 0,C 180,E1 -24471.559,E2 -24471.559} C_VEL
LIN {X 0,Y 144.158,Z 180.514,A -85,B 0,C 180,E1 -24480.002,E2 -24480.002} C_VEL
LIN {X 0,Y 143.61,Z 180.583,A -85,B 0,C 180,E1 -24488.444,E2 -24488.444} C_VEL
LIN {X 0,Y 143.502,Z 180.611,A -85,B 0,C 180,E1 -24491.616,E2 -24491.616} C_VEL
LIN {X 0,Y 143.257,Z 180.629,A -85,B 0,C 180,E1 -24497.12,E2 -24497.12} C_VEL
LIN {X 0,Y 143.226,Z 180.643,A -85,B 0,C 180,E1 -24501.199,E2 -24501.199} C_VEL
LIN {X 0,Y 143.187,Z 180.648,A -85,B 0,C 180,E1 -24507.932,E2 -24507.932} C_VEL
LIN {X 0,Y 143.142,Z 180.656,A -85,B 0,C 180,E1 -24513.417,E2 -24513.417} C_VEL
LIN {X 0,Y 143.056,Z 180.669,A -85,B 0,C 180,E1 -24519.694,E2 -24519.694} C_VEL
LIN {X 0,Y 143.106,Z 180.752,A -85,B 0,C 180,E1 -24521.725,E2 -24521.725} C_VEL
LIN {X 0,Y 144.086,Z 183.514,A -85,B 0,C 180,E1 -24522.233,E2 -24522.233} C_VEL
LIN {X 0,Y 145.831,Z 185.74,A -85,B 0,C 180,E1 -24522.939,E2 -24522.939} C_VEL
LIN {X 0,Y 149.697,Z 192.396,A -85,B 0,C 180,E1 -24524.532,E2 -24524.532} C_VEL
LIN {X 0,Y 156.035,Z 206.377,A -85,B 0,C 180,E1 -24527.085,E2 -24527.085} C_VEL
LIN {X 0,Y 161.238,Z 220.485,A -85,B 0,C 180,E1 -24529.139,E2 -24529.139} C_VEL
LIN {X 0,Y 162.662,Z 225.103,A -85,B 0,C 180,E1 -24529.713,E2 -24529.713} C_VEL
LIN {X 0,Y 164.231,Z 243.381,A -85,B 0,C 180,E1 -24531.017,E2 -24531.017} C_VEL
LIN {X 0,Y 161.698,Z 288.448,A -85,B 0,C 180,E1 -24532.91,E2 -24532.91} C_VEL
LIN {X 0,Y 160.09,Z 302.338,A -85,B 0,C 180,E1 -24533.946,E2 -24533.946} C_VEL
LIN {X 0,Y 158.113,Z 314.284,A -85,B 0,C 180,E1 -24535.283,E2 -24535.283} C_VEL
LIN {X 0,Y 155.961,Z 324.769,A -85,B 0,C 180,E1 -24536.88,E2 -24536.88} C_VEL
LIN {X 0,Y 153.037,Z 336.665,A -85,B 0,C 180,E1 -24539.275,E2 -24539.275} C_VEL
LIN {X 0,Y 150.428,Z 346.237,A -85,B 0,C 180,E1 -24541.767,E2 -24541.767} C_VEL
LIN {X 0,Y 147.919,Z 355.129,A -85,B 0,C 180,E1 -24544.683,E2 -24544.683} C_VEL
LIN {X 0,Y 145.587,Z 363.294,A -85,B 0,C 180,E1 -24548.029,E2 -24548.029} C_VEL
LIN {X 0,Y 143.374,Z 371.27,A -85,B 0,C 180,E1 -24552.159,E2 -24552.159} C_VEL
LIN {X 0,Y 142.046,Z 376.661,A -85,B 0,C 180,E1 -24555.677,E2 -24555.677} C_VEL
LIN {X 0,Y 141.099,Z 381.902,A -85,B 0,C 180,E1 -24559.96,E2 -24559.96} C_VEL
LIN {X 0,Y 140.698,Z 385.935,A -85,B 0,C 180,E1 -24564.266,E2 -24564.266} C_VEL
LIN {X 0,Y 140.669,Z 388.392,A -85,B 0,C 180,E1 -24567.78,E2 -24567.78} C_VEL
LIN {X 0,Y 140.775,Z 389.383,A -85,B 0,C 180,E1 -24569.576,E2 -24569.576} C_VEL
LIN {X 0,Y 140.561,Z 390.162,A -85,B 0,C 180,E1 -24571.137,E2 -24571.137} C_VEL
LIN {X 0,Y 139.785,Z 390.779,A -85,B 0,C 180,E1 -24572.692,E2 -24572.692} C_VEL
LIN {X 0,Y 137.382,Z 391.561,A -85,B 0,C 180,E1 -24575.81,E2 -24575.81} C_VEL
LIN {X 0,Y 135.088,Z 391.811,A -85,B 0,C 180,E1 -24579.063,E2 -24579.063} C_VEL
LIN {X 0,Y 134.414,Z 391.701,A -85,B 0,C 180,E1 -24581.599,E2 -24581.599} C_VEL
LIN {X 0,Y 134.527,Z 391.613,A -85,B 0,C 180,E1 -24582.449,E2 -24582.449} C_VEL
LIN {X 0,Y 136.558,Z 390.573,A -85,B 0,C 180,E1 -24587.986,E2 -24587.986} C_VEL
LIN {X 0,Y 138.248,Z 389.47,A -85,B 0,C 180,E1 -24590.845,E2 -24590.845} C_VEL
LIN {X 0,Y 140.32,Z 387.935,A -85,B 0,C 180,E1 -24593.621,E2 -24593.621} C_VEL
LIN {X 0,Y 143.96,Z 384.88,A -85,B 0,C 180,E1 -24597.631,E2 -24597.631} C_VEL
LIN {X 0,Y 148.155,Z 380.817,A -85,B 0,C 180,E1 -24601.453,E2 -24601.453} C_VEL
LIN {X 0,Y 154.014,Z 374.626,A -85,B 0,C 180,E1 -24605.578,E2 -24605.578} C_VEL
LIN {X 0,Y 159.743,Z 367.924,A -85,B 0,C 180,E1 -24608.824,E2 -24608.824} C_VEL
LIN {X 0,Y 165.968,Z 359.653,A -85,B 0,C 180,E1 -24611.831,E2 -24611.831} C_VEL
LIN {X 0,Y 171.491,Z 351.197,A -85,B 0,C 180,E1 -24614.162,E2 -24614.162} C_VEL
LIN {X 0,Y 177.408,Z 340.786,A -85,B 0,C 180,E1 -24616.3,E2 -24616.3} C_VEL
LIN {X 0,Y 182.334,Z 330.524,A -85,B 0,C 180,E1 -24617.9,E2 -24617.9} C_VEL
LIN {X 0,Y 186.814,Z 319.309,A -85,B 0,C 180,E1 -24619.21,E2 -24619.21} C_VEL
LIN {X 0,Y 190.406,Z 307.932,A -85,B 0,C 180,E1 -24620.192,E2 -24620.192} C_VEL
LIN {X 0,Y 193.426,Z 294.855,A -85,B 0,C 180,E1 -24620.974,E2 -24620.974} C_VEL
LIN {X 0,Y 195.233,Z 281.633,A -85,B 0,C 180,E1 -24621.538,E2 -24621.538} C_VEL
LIN {X 0,Y 196.696,Z 264.1,A -85,B 0,C 180,E1 -24622.113,E2 -24622.113} C_VEL
LIN {X 0,Y 193.05,Z 254.597,A -85,B 0,C 180,E1 -24624.853,E2 -24624.853} C_VEL
LIN {X 0,Y 189.379,Z 246.385,A -85,B 0,C 180,E1 -24627.914,E2 -24627.914} C_VEL
LIN {X 0,Y 186.323,Z 239.938,A -85,B 0,C 180,E1 -24630.849,E2 -24630.849} C_VEL
LIN {X 0,Y 183.552,Z 234.628,A -85,B 0,C 180,E1 -24634.027,E2 -24634.027} C_VEL
LIN {X 0,Y 181.045,Z 230.029,A -85,B 0,C 180,E1 -24637.609,E2 -24637.609} C_VEL
LIN {X 0,Y 179.625,Z 227.955,A -85,B 0,C 180,E1 -24640.08,E2 -24640.08} C_VEL
LIN {X 0,Y 178.091,Z 224.722,A -85,B 0,C 180,E1 -24644.291,E2 -24644.291} C_VEL
LIN {X 0,Y 177.847,Z 224.249,A -85,B 0,C 180,E1 -24645.262,E2 -24645.262} C_VEL
LIN {X 0,Y 177.282,Z 223.877,A -85,B 0,C 180,E1 -24652.339,E2 -24652.339} C_VEL
LIN {X 0,Y 178.476,Z 224.468,A -85,B 0,C 180,E1 -24657.209,E2 -24657.209} C_VEL
LIN {X 0,Y 179.683,Z 227.538,A -85,B 0,C 180,E1 -24660.485,E2 -24660.485} C_VEL
LIN {X 0,Y 181.422,Z 229.503,A -85,B 0,C 180,E1 -24663.341,E2 -24663.341} C_VEL
LIN {X 0,Y 184.156,Z 233.944,A -85,B 0,C 180,E1 -24667.029,E2 -24667.029} C_VEL
LIN {X 0,Y 187.125,Z 238.705,A -85,B 0,C 180,E1 -24670.209,E2 -24670.209} C_VEL
LIN {X 0,Y 191.036,Z 245.213,A -85,B 0,C 180,E1 -24673.631,E2 -24673.631} C_VEL
LIN {X 0,Y 194.977,Z 252.411,A -85,B 0,C 180,E1 -24676.616,E2 -24676.616} C_VEL
LIN {X 0,Y 197.313,Z 257.127,A -85,B 0,C 180,E1 -24678.234,E2 -24678.234} C_VEL
LIN {X 0,Y 195.055,Z 280.988,A -85,B 0,C 180,E1 -24679.022,E2 -24679.022} C_VEL
LIN {X 0,Y 192.671,Z 294.257,A -85,B 0,C 180,E1 -24679.729,E2 -24679.729} C_VEL
LIN {X 0,Y 189.671,Z 305.987,A -85,B 0,C 180,E1 -24680.674,E2 -24680.674} C_VEL
LIN {X 0,Y 185.466,Z 318.383,A -85,B 0,C 180,E1 -24682.073,E2 -24682.073} C_VEL
LIN {X 0,Y 180.468,Z 329.892,A -85,B 0,C 180,E1 -24683.771,E2 -24683.771} C_VEL
LIN {X 0,Y 175.455,Z 339.574,A -85,B 0,C 180,E1 -24685.679,E2 -24685.679} C_VEL
LIN {X 0,Y 169.442,Z 349.304,A -85,B 0,C 180,E1 -24688.189,E2 -24688.189} C_VEL
LIN {X 0,Y 163.357,Z 357.765,A -85,B 0,C 180,E1 -24691.081,E2 -24691.081} C_VEL
LIN {X 0,Y 157.477,Z 364.894,A -85,B 0,C 180,E1 -24694.348,E2 -24694.348} C_VEL
LIN {X 0,Y 151.794,Z 370.857,A -85,B 0,C 180,E1 -24698.086,E2 -24698.086} C_VEL
LIN {X 0,Y 146.868,Z 375.406,A -85,B 0,C 180,E1 -24702.06,E2 -24702.06} C_VEL
LIN {X 0,Y 142.581,Z 378.801,A -85,B 0,C 180,E1 -24706.364,E2 -24706.364} C_VEL
LIN {X 0,Y 140.209,Z 380.424,A -85,B 0,C 180,E1 -24709.336,E2 -24709.336} C_VEL
LIN {X 0,Y 138.177,Z 381.528,A -85,B 0,C 180,E1 -24712.386,E2 -24712.386} C_VEL
LIN {X 0,Y 136.528,Z 382.177,A -85,B 0,C 180,E1 -24715.512,E2 -24715.512} C_VEL
LIN {X 0,Y 135.176,Z 382.399,A -85,B 0,C 180,E1 -24718.674,E2 -24718.674} C_VEL
LIN {X 0,Y 133.95,Z 381.915,A -85,B 0,C 180,E1 -24723.115,E2 -24723.115} C_VEL
LIN {X 0,Y 133.211,Z 380.294,A -85,B 0,C 180,E1 -24728.327,E2 -24728.327} C_VEL
LIN {X 0,Y 133.206,Z 378.554,A -85,B 0,C 180,E1 -24731.742,E2 -24731.742} C_VEL
LIN {X 0,Y 133.636,Z 375.386,A -85,B 0,C 180,E1 -24736.311,E2 -24736.311} C_VEL
LIN {X 0,Y 134.638,Z 370.975,A -85,B 0,C 180,E1 -24740.991,E2 -24740.991} C_VEL
LIN {X 0,Y 136.087,Z 365.348,A -85,B 0,C 180,E1 -24745.558,E2 -24745.558} C_VEL
LIN {X 0,Y 138.157,Z 358.311,A -85,B 0,C 180,E1 -24750.001,E2 -24750.001} C_VEL
LIN {X 0,Y 140.689,Z 350.299,A -85,B 0,C 180,E1 -24753.946,E2 -24753.946} C_VEL
LIN {X 0,Y 143.667,Z 340.41,A -85,B 0,C 180,E1 -24757.732,E2 -24757.732} C_VEL
LIN {X 0,Y 146.537,Z 330.416,A -85,B 0,C 180,E1 -24760.711,E2 -24760.711} C_VEL
LIN {X 0,Y 149.333,Z 319.393,A -85,B 0,C 180,E1 -24763.264,E2 -24763.264} C_VEL
LIN {X 0,Y 151.729,Z 308.043,A -85,B 0,C 180,E1 -24765.275,E2 -24765.275} C_VEL
LIN {X 0,Y 154.005,Z 295.081,A -85,B 0,C 180,E1 -24766.948,E2 -24766.948} C_VEL
LIN {X 0,Y 155.465,Z 282.662,A -85,B 0,C 180,E1 -24768.064,E2 -24768.064} C_VEL
LIN {X 0,Y 156.613,Z 266.64,A -85,B 0,C 180,E1 -24768.885,E2 -24768.885} C_VEL
LIN {X 0,Y 159.173,Z 224.889,A -85,B 0,C 180,E1 -24770.587,E2 -24770.587} C_VEL
LIN {X 0,Y 152.08,Z 209.438,A -85,B 0,C 180,E1 -24773.253,E2 -24773.253} C_VEL
LIN {X 0,Y 146.621,Z 199.272,A -85,B 0,C 180,E1 -24775.429,E2 -24775.429} C_VEL
LIN {X 0,Y 140.457,Z 189.257,A -85,B 0,C 180,E1 -24778.08,E2 -24778.08} C_VEL
LIN {X 0,Y 138.36,Z 185.931,A -85,B 0,C 180,E1 -24779.053,E2 -24779.053} C_VEL
LIN {X 0,Y 136.578,Z 183.523,A -85,B 0,C 180,E1 -24779.876,E2 -24779.876} C_VEL
LIN {X 0,Y 136.038,Z 181.528,A -85,B 0,C 180,E1 -24780.239,E2 -24780.239} C_VEL
LIN {X 0,Y 136.036,Z 181.518,A -85,B 0,C 180,E1 -24784.632,E2 -24784.632} C_VEL
LIN {X 0,Y 136.022,Z 181.534,A -85,B 0,C 180,E1 -24789.196,E2 -24789.196} C_VEL
LIN {X 0,Y 135.976,Z 181.527,A -85,B 0,C 180,E1 -24793.65,E2 -24793.65} C_VEL
LIN {X 0,Y 135.98,Z 181.505,A -85,B 0,C 180,E1 -24797.789,E2 -24797.789} C_VEL
LIN {X 0,Y 136.02,Z 181.537,A -85,B 0,C 180,E1 -24801.684,E2 -24801.684} C_VEL
LIN {X 0,Y 136.051,Z 181.521,A -85,B 0,C 180,E1 -24805.744,E2 -24805.744} C_VEL
LIN {X 0,Y 136.085,Z 181.481,A -85,B 0,C 180,E1 -24812.305,E2 -24812.305} C_VEL
LIN {X 0,Y 136.182,Z 181.521,A -85,B 0,C 180,E1 -24818.825,E2 -24818.825} C_VEL
LIN {X 0,Y 136.223,Z 181.513,A -85,B 0,C 180,E1 -24825.053,E2 -24825.053} C_VEL
LIN {X 0,Y 136.427,Z 181.489,A -85,B 0,C 180,E1 -24828.18,E2 -24828.18} C_VEL
LIN {X 0,Y 136.537,Z 181.461,A -85,B 0,C 180,E1 -24831.119,E2 -24831.119} C_VEL
LIN {X 0,Y 137.115,Z 181.391,A -85,B 0,C 180,E1 -24840.002,E2 -24840.002} C_VEL
LIN {X 0,Y 136.539,Z 181.464,A -85,B 0,C 180,E1 -24848.885,E2 -24848.885} C_VEL
LIN {X 0,Y 136.417,Z 181.495,A -85,B 0,C 180,E1 -24851.894,E2 -24851.894} C_VEL
LIN {X 0,Y 136.17,Z 181.517,A -85,B 0,C 180,E1 -24858.041,E2 -24858.041} C_VEL
LIN {X 0,Y 136.152,Z 181.523,A -85,B 0,C 180,E1 -24861.697,E2 -24861.697} C_VEL
LIN {X 0,Y 136.096,Z 181.532,A -85,B 0,C 180,E1 -24868.611,E2 -24868.611} C_VEL
LIN {X 0,Y 136.044,Z 181.54,A -85,B 0,C 180,E1 -24874.631,E2 -24874.631} C_VEL
LIN {X 0,Y 136.007,Z 181.548,A -85,B 0,C 180,E1 -24879.184,E2 -24879.184} C_VEL
LIN {X 0,Y 137.064,Z 184.439,A -85,B 0,C 180,E1 -24879.845,E2 -24879.845} C_VEL
LIN {X 0,Y 138.963,Z 186.876,A -85,B 0,C 180,E1 -24880.708,E2 -24880.708} C_VEL
LIN {X 0,Y 144.492,Z 195.895,A -85,B 0,C 180,E1 -24883.173,E2 -24883.173} C_VEL
LIN {X 0,Y 150.741,Z 209.83,A -85,B 0,C 180,E1 -24885.881,E2 -24885.881} C_VEL
LIN {X 0,Y 155.69,Z 223.486,A -85,B 0,C 180,E1 -24887.968,E2 -24887.968} C_VEL
LIN {X 0,Y 156.816,Z 227.16,A -85,B 0,C 180,E1 -24888.454,E2 -24888.454} C_VEL
LIN {X 0,Y 158.185,Z 243.862,A -85,B 0,C 180,E1 -24889.706,E2 -24889.706} C_VEL
LIN {X 0,Y 155.479,Z 289.08,A -85,B 0,C 180,E1 -24891.674,E2 -24891.674} C_VEL
LIN {X 0,Y 153.787,Z 302.667,A -85,B 0,C 180,E1 -24892.733,E2 -24892.733} C_VEL
LIN {X 0,Y 151.865,Z 313.909,A -85,B 0,C 180,E1 -24894.044,E2 -24894.044} C_VEL
LIN {X 0,Y 149.637,Z 324.426,A -85,B 0,C 180,E1 -24895.694,E2 -24895.694} C_VEL
LIN {X 0,Y 146.564,Z 336.339,A -85,B 0,C 180,E1 -24898.165,E2 -24898.165} C_VEL
LIN {X 0,Y 143.819,Z 345.92,A -85,B 0,C 180,E1 -24900.746,E2 -24900.746} C_VEL
LIN {X 0,Y 141.501,Z 353.925,A -85,B 0,C 180,E1 -24903.447,E2 -24903.447} C_VEL
LIN {X 0,Y 139.473,Z 360.739,A -85,B 0,C 180,E1 -24906.226,E2 -24906.226} C_VEL
LIN {X 0,Y 137.01,Z 369.137,A -85,B 0,C 180,E1 -24910.523,E2 -24910.523} C_VEL
LIN {X 0,Y 135.122,Z 375.864,A -85,B 0,C 180,E1 -24914.926,E2 -24914.926} C_VEL
LIN {X 0,Y 134.085,Z 381.221,A -85,B 0,C 180,E1 -24919.429,E2 -24919.429} C_VEL
LIN {X 0,Y 133.631,Z 385.354,A -85,B 0,C 180,E1 -24923.962,E2 -24923.962} C_VEL
LIN {X 0,Y 133.614,Z 388.119,A -85,B 0,C 180,E1 -24928.037,E2 -24928.037} C_VEL
LIN {X 0,Y 133.723,Z 389.166,A -85,B 0,C 180,E1 -24929.999,E2 -24929.999} C_VEL
LIN {X 0,Y 133.569,Z 390.391,A -85,B 0,C 180,E1 -24933.016,E2 -24933.016} C_VEL
LIN {X 0,Y 133.554,Z 391.219,A -85,B 0,C 180,E1 -24936.041,E2 -24936.041} C_VEL
LIN {X 0,Y 133.855,Z 391.643,A -85,B 0,C 180,E1 -24939.062,E2 -24939.062} C_VEL
LIN {X 0,Y 134.527,Z 391.613,A -85,B 0,C 180,E1 -24942.449,E2 -24942.449} C_VEL
LIN {X 0,Y 134.639,Z 391.326,A -85,B 0,C 180,E1 -24944.959,E2 -24944.959} C_VEL
LIN {X 0,Y 133.633,Z 390.296,A -85,B 0,C 180,E1 -24949.154,E2 -24949.154} C_VEL
LIN {X 0,Y 133.352,Z 388.691,A -85,B 0,C 180,E1 -24953.345,E2 -24953.345} C_VEL
LIN {X 0,Y 134.564,Z 387.324,A -85,B 0,C 180,E1 -24955.743,E2 -24955.743} C_VEL
LIN {X 0,Y 139.14,Z 383.717,A -85,B 0,C 180,E1 -24960.338,E2 -24960.338} C_VEL
LIN {X 0,Y 143.784,Z 379.396,A -85,B 0,C 180,E1 -24964.201,E2 -24964.201} C_VEL
LIN {X 0,Y 150.226,Z 372.917,A -85,B 0,C 180,E1 -24968.307,E2 -24968.307} C_VEL
LIN {X 0,Y 156.45,Z 365.847,A -85,B 0,C 180,E1 -24971.498,E2 -24971.498} C_VEL
LIN {X 0,Y 163.077,Z 357.087,A -85,B 0,C 180,E1 -24974.452,E2 -24974.452} C_VEL
LIN {X 0,Y 169.522,Z 347.181,A -85,B 0,C 180,E1 -24976.944,E2 -24976.944} C_VEL
LIN {X 0,Y 175.135,Z 337.101,A -85,B 0,C 180,E1 -24978.8,E2 -24978.8} C_VEL
LIN {X 0,Y 180.325,Z 325.966,A -85,B 0,C 180,E1 -24980.33,E2 -24980.33} C_VEL
LIN {X 0,Y 184.968,Z 313.535,A -85,B 0,C 180,E1 -24981.597,E2 -24981.597} C_VEL
LIN {X 0,Y 188.624,Z 300.587,A -85,B 0,C 180,E1 -24982.489,E2 -24982.489} C_VEL
LIN {X 0,Y 191.063,Z 287.329,A -85,B 0,C 180,E1 -24983.156,E2 -24983.156} C_VEL
LIN {X 0,Y 193.041,Z 267.204,A -85,B 0,C 180,E1 -24983.817,E2 -24983.817} C_VEL
LIN {X 0,Y 189.976,Z 258.967,A -85,B 0,C 180,E1 -24986.351,E2 -24986.351} C_VEL
LIN {X 0,Y 186.801,Z 251.466,A -85,B 0,C 180,E1 -24989.251,E2 -24989.251} C_VEL
LIN {X 0,Y 183.849,Z 245.08,A -85,B 0,C 180,E1 -24992.385,E2 -24992.385} C_VEL
LIN {X 0,Y 181.909,Z 241.052,A -85,B 0,C 180,E1 -24994.849,E2 -24994.849} C_VEL
LIN {X 0,Y 179.73,Z 236.763,A -85,B 0,C 180,E1 -24998.192,E2 -24998.192} C_VEL
LIN {X 0,Y 178.338,Z 234.662,A -85,B 0,C 180,E1 -25000.789,E2 -25000.789} C_VEL
LIN {X 0,Y 176.96,Z 231.318,A -85,B 0,C 180,E1 -25005.187,E2 -25005.187} C_VEL
LIN {X 0,Y 176.26,Z 230.842,A -85,B 0,C 180,E1 -25010.821,E2 -25010.821} C_VEL
LIN {X 0,Y 177.407,Z 231.449,A -85,B 0,C 180,E1 -25016.765,E2 -25016.765} C_VEL
LIN {X 0,Y 178.746,Z 234.735,A -85,B 0,C 180,E1 -25020.487,E2 -25020.487} C_VEL
LIN {X 0,Y 180.145,Z 236.419,A -85,B 0,C 180,E1 -25022.865,E2 -25022.865} C_VEL
LIN {X 0,Y 182.564,Z 240.474,A -85,B 0,C 180,E1 -25026.307,E2 -25026.307} C_VEL
LIN {X 0,Y 185.35,Z 245.219,A -85,B 0,C 180,E1 -25029.496,E2 -25029.496} C_VEL
LIN {X 0,Y 188.963,Z 251.485,A -85,B 0,C 180,E1 -25032.839,E2 -25032.839} C_VEL
LIN {X 0,Y 193.018,Z 259.31,A -85,B 0,C 180,E1 -25036.069,E2 -25036.069} C_VEL
LIN {X 0,Y 193.54,Z 260.381,A -85,B 0,C 180,E1 -25036.455,E2 -25036.455} C_VEL
LIN {X 0,Y 191.574,Z 281.103,A -85,B 0,C 180,E1 -25037.195,E2 -25037.195} C_VEL
LIN {X 0,Y 189.221,Z 293.837,A -85,B 0,C 180,E1 -25037.848,E2 -25037.848} C_VEL
LIN {X 0,Y 186.269,Z 305.186,A -85,B 0,C 180,E1 -25038.727,E2 -25038.727} C_VEL
LIN {X 0,Y 182.22,Z 317.111,A -85,B 0,C 180,E1 -25040.012,E2 -25040.012} C_VEL
LIN {X 0,Y 177.536,Z 327.856,A -85,B 0,C 180,E1 -25041.522,E2 -25041.522} C_VEL
LIN {X 0,Y 172.283,Z 337.923,A -85,B 0,C 180,E1 -25043.386,E2 -25043.386} C_VEL
LIN {X 0,Y 167.118,Z 346.303,A -85,B 0,C 180,E1 -25045.361,E2 -25045.361} C_VEL
LIN {X 0,Y 161.146,Z 354.773,A -85,B 0,C 180,E1 -25047.975,E2 -25047.975} C_VEL
LIN {X 0,Y 154.336,Z 362.977,A -85,B 0,C 180,E1 -25051.37,E2 -25051.37} C_VEL
LIN {X 0,Y 149.04,Z 368.527,A -85,B 0,C 180,E1 -25054.46,E2 -25054.46} C_VEL
LIN {X 0,Y 143.485,Z 373.695,A -85,B 0,C 180,E1 -25058.4,E2 -25058.4} C_VEL
LIN {X 0,Y 138.563,Z 377.622,A -85,B 0,C 180,E1 -25062.655,E2 -25062.655} C_VEL
LIN {X 0,Y 134.44,Z 380.372,A -85,B 0,C 180,E1 -25067.189,E2 -25067.189} C_VEL
LIN {X 0,Y 132.132,Z 381.616,A -85,B 0,C 180,E1 -25070.337,E2 -25070.337} C_VEL
LIN {X 0,Y 129.947,Z 382.433,A -85,B 0,C 180,E1 -25074.216,E2 -25074.216} C_VEL
LIN {X 0,Y 127.488,Z 382.507,A -85,B 0,C 180,E1 -25080.255,E2 -25080.255} C_VEL
LIN {X 0,Y 126.704,Z 381.878,A -85,B 0,C 180,E1 -25083.658,E2 -25083.658} C_VEL
LIN {X 0,Y 126.211,Z 380.821,A -85,B 0,C 180,E1 -25087.059,E2 -25087.059} C_VEL
LIN {X 0,Y 126.084,Z 378.836,A -85,B 0,C 180,E1 -25091.362,E2 -25091.362} C_VEL
LIN {X 0,Y 126.676,Z 374.894,A -85,B 0,C 180,E1 -25097.179,E2 -25097.179} C_VEL
LIN {X 0,Y 127.762,Z 370.434,A -85,B 0,C 180,E1 -25101.941,E2 -25101.941} C_VEL
LIN {X 0,Y 129.486,Z 364.401,A -85,B 0,C 180,E1 -25106.889,E2 -25106.889} C_VEL
LIN {X 0,Y 131.769,Z 357.026,A -85,B 0,C 180,E1 -25111.529,E2 -25111.529} C_VEL
LIN {X 0,Y 134.747,Z 347.838,A -85,B 0,C 180,E1 -25115.988,E2 -25115.988} C_VEL
LIN {X 0,Y 137.804,Z 338.338,A -85,B 0,C 180,E1 -25119.541,E2 -25119.541} C_VEL
LIN {X 0,Y 140.879,Z 327.739,A -85,B 0,C 180,E1 -25122.607,E2 -25122.607} C_VEL
LIN {X 0,Y 143.927,Z 315.944,A -85,B 0,C 180,E1 -25125.217,E2 -25125.217} C_VEL
LIN {X 0,Y 146.28,Z 304.409,A -85,B 0,C 180,E1 -25127.151,E2 -25127.151} C_VEL
LIN {X 0,Y 148.424,Z 291.255,A -85,B 0,C 180,E1 -25128.713,E2 -25128.713} C_VEL
LIN {X 0,Y 149.896,Z 278.07,A -85,B 0,C 180,E1 -25129.744,E2 -25129.744} C_VEL
LIN {X 0,Y 153.03,Z 226.524,A -85,B 0,C 180,E1 -25132.004,E2 -25132.004} C_VEL
LIN {X 0,Y 145.743,Z 210.689,A -85,B 0,C 180,E1 -25134.971,E2 -25134.971} C_VEL
LIN {X 0,Y 138.992,Z 198.601,A -85,B 0,C 180,E1 -25137.946,E2 -25137.946} C_VEL
LIN {X 0,Y 134.055,Z 190.916,A -85,B 0,C 180,E1 -25140.303,E2 -25140.303} C_VEL
LIN {X 0,Y 131.967,Z 187.565,A -85,B 0,C 180,E1 -25141.381,E2 -25141.381} C_VEL
LIN {X 0,Y 129.733,Z 184.847,A -85,B 0,C 180,E1 -25142.528,E2 -25142.528} C_VEL
LIN {X 0,Y 128.982,Z 182.412,A -85,B 0,C 180,E1 -25143.15,E2 -25143.15} C_VEL
LIN {X 0,Y 128.92,Z 182.398,A -85,B 0,C 180,E1 -25146.846,E2 -25146.846} C_VEL
LIN {X 0,Y 128.92,Z 182.427,A -85,B 0,C 180,E1 -25150.858,E2 -25150.858} C_VEL
LIN {X 0,Y 128.91,Z 182.388,A -85,B 0,C 180,E1 -25155.134,E2 -25155.134} C_VEL
LIN {X 0,Y 128.932,Z 182.401,A -85,B 0,C 180,E1 -25159.742,E2 -25159.742} C_VEL
LIN {X 0,Y 128.955,Z 182.413,A -85,B 0,C 180,E1 -25164.836,E2 -25164.836} C_VEL
LIN {X 0,Y 128.982,Z 182.355,A -85,B 0,C 180,E1 -25170.672,E2 -25170.672} C_VEL
LIN {X 0,Y 129.067,Z 182.407,A -85,B 0,C 180,E1 -25177.775,E2 -25177.775} C_VEL
LIN {X 0,Y 129.145,Z 182.388,A -85,B 0,C 180,E1 -25184.213,E2 -25184.213} C_VEL
LIN {X 0,Y 129.345,Z 182.372,A -85,B 0,C 180,E1 -25187.975,E2 -25187.975} C_VEL
LIN {X 0,Y 129.463,Z 182.342,A -85,B 0,C 180,E1 -25190.629,E2 -25190.629} C_VEL
LIN {X 0,Y 130.07,Z 182.268,A -85,B 0,C 180,E1 -25200.002,E2 -25200.002} C_VEL
LIN {X 0,Y 129.465,Z 182.347,A -85,B 0,C 180,E1 -25209.374,E2 -25209.374} C_VEL
LIN {X 0,Y 129.3,Z 182.38,A -85,B 0,C 180,E1 -25212.559,E2 -25212.559} C_VEL
LIN {X 0,Y 129.088,Z 182.404,A -85,B 0,C 180,E1 -25219.068,E2 -25219.068} C_VEL
LIN {X 0,Y 129.049,Z 182.408,A -85,B 0,C 180,E1 -25222.411,E2 -25222.411} C_VEL
LIN {X 0,Y 129.021,Z 182.414,A -85,B 0,C 180,E1 -25229.359,E2 -25229.359} C_VEL
LIN {X 0,Y 128.96,Z 182.424,A -85,B 0,C 180,E1 -25235.167,E2 -25235.167} C_VEL
LIN {X 0,Y 128.934,Z 182.426,A -85,B 0,C 180,E1 -25236.357,E2 -25236.357} C_VEL
LIN {X 0,Y 129.861,Z 185.145,A -85,B 0,C 180,E1 -25237.021,E2 -25237.021} C_VEL
LIN {X 0,Y 132.006,Z 187.702,A -85,B 0,C 180,E1 -25238.118,E2 -25238.118} C_VEL
LIN {X 0,Y 134.093,Z 191.003,A -85,B 0,C 180,E1 -25239.193,E2 -25239.193} C_VEL
LIN {X 0,Y 139.329,Z 199.335,A -85,B 0,C 180,E1 -25241.7,E2 -25241.7} C_VEL
LIN {X 0,Y 145.196,Z 212.512,A -85,B 0,C 180,E1 -25244.456,E2 -25244.456} C_VEL
LIN {X 0,Y 150.208,Z 226.501,A -85,B 0,C 180,E1 -25246.733,E2 -25246.733} C_VEL
LIN {X 0,Y 151.027,Z 229.617,A -85,B 0,C 180,E1 -25247.134,E2 -25247.134} C_VEL
LIN {X 0,Y 152.205,Z 244.974,A -85,B 0,C 180,E1 -25248.327,E2 -25248.327} C_VEL
LIN {X 0,Y 149.45,Z 288.55,A -85,B 0,C 180,E1 -25250.263,E2 -25250.263} C_VEL
LIN {X 0,Y 147.702,Z 302.235,A -85,B 0,C 180,E1 -25251.352,E2 -25251.352} C_VEL
LIN {X 0,Y 145.695,Z 313.522,A -85,B 0,C 180,E1 -25252.699,E2 -25252.699} C_VEL
LIN {X 0,Y 143.365,Z 324.069,A -85,B 0,C 180,E1 -25254.398,E2 -25254.398} C_VEL
LIN {X 0,Y 140.157,Z 336.01,A -85,B 0,C 180,E1 -25256.953,E2 -25256.953} C_VEL
LIN {X 0,Y 136.981,Z 346.697,A -85,B 0,C 180,E1 -25259.983,E2 -25259.983} C_VEL
LIN {X 0,Y 134.627,Z 354.202,A -85,B 0,C 180,E1 -25262.671,E2 -25262.671} C_VEL
LIN {X 0,Y 131.932,Z 362.701,A -85,B 0,C 180,E1 -25266.451,E2 -25266.451} C_VEL
LIN {X 0,Y 129.48,Z 370.695,A -85,B 0,C 180,E1 -25270.993,E2 -25270.993} C_VEL
LIN {X 0,Y 127.776,Z 377.046,A -85,B 0,C 180,E1 -25275.669,E2 -25275.669} C_VEL
LIN {X 0,Y 126.854,Z 382.077,A -85,B 0,C 180,E1 -25280.432,E2 -25280.432} C_VEL
LIN {X 0,Y 126.48,Z 385.927,A -85,B 0,C 180,E1 -25285.218,E2 -25285.218} C_VEL
LIN {X 0,Y 126.636,Z 388.713,A -85,B 0,C 180,E1 -25289.999,E2 -25289.999} C_VEL
LIN {X 0,Y 126.493,Z 389.98,A -85,B 0,C 180,E1 -25293.184,E2 -25293.184} C_VEL
LIN {X 0,Y 126.843,Z 391.34,A -85,B 0,C 180,E1 -25299.568,E2 -25299.568} C_VEL
LIN {X 0,Y 128.458,Z 391.107,A -85,B 0,C 180,E1 -25305.875,E2 -25305.875} C_VEL
LIN {X 0,Y 131.616,Z 389.371,A -85,B 0,C 180,E1 -25311.949,E2 -25311.949} C_VEL
LIN {X 0,Y 134.564,Z 387.324,A -85,B 0,C 180,E1 -25315.743,E2 -25315.743} C_VEL
LIN {X 0,Y 135.987,Z 385.813,A -85,B 0,C 180,E1 -25318.081,E2 -25318.081} C_VEL
LIN {X 0,Y 137.079,Z 382.889,A -85,B 0,C 180,E1 -25322.044,E2 -25322.044} C_VEL
LIN {X 0,Y 138.737,Z 379.407,A -85,B 0,C 180,E1 -25325.835,E2 -25325.835} C_VEL
LIN {X 0,Y 140.954,Z 376.884,A -85,B 0,C 180,E1 -25327.821,E2 -25327.821} C_VEL
LIN {X 0,Y 147.893,Z 369.958,A -85,B 0,C 180,E1 -25331.705,E2 -25331.705} C_VEL
LIN {X 0,Y 154.58,Z 362.288,A -85,B 0,C 180,E1 -25334.806,E2 -25334.806} C_VEL
LIN {X 0,Y 161.696,Z 352.728,A -85,B 0,C 180,E1 -25337.637,E2 -25337.637} C_VEL
LIN {X 0,Y 167.989,Z 342.897,A -85,B 0,C 180,E1 -25339.774,E2 -25339.774} C_VEL
LIN {X 0,Y 173.893,Z 331.879,A -85,B 0,C 180,E1 -25341.541,E2 -25341.541} C_VEL
LIN {X 0,Y 179.333,Z 319.382,A -85,B 0,C 180,E1 -25342.986,E2 -25342.986} C_VEL
LIN {X 0,Y 183.253,Z 307.854,A -85,B 0,C 180,E1 -25343.956,E2 -25343.956} C_VEL
LIN {X 0,Y 186.396,Z 295.292,A -85,B 0,C 180,E1 -25344.689,E2 -25344.689} C_VEL
LIN {X 0,Y 188.457,Z 281.613,A -85,B 0,C 180,E1 -25345.271,E2 -25345.271} C_VEL
LIN {X 0,Y 189.517,Z 270.137,A -85,B 0,C 180,E1 -25345.645,E2 -25345.645} C_VEL
LIN {X 0,Y 186.585,Z 262.137,A -85,B 0,C 180,E1 -25348.332,E2 -25348.332} C_VEL
LIN {X 0,Y 183.552,Z 254.732,A -85,B 0,C 180,E1 -25351.481,E2 -25351.481} C_VEL
LIN {X 0,Y 180.703,Z 248.147,A -85,B 0,C 180,E1 -25355.136,E2 -25355.136} C_VEL
LIN {X 0,Y 178.351,Z 243.394,A -85,B 0,C 180,E1 -25358.925,E2 -25358.925} C_VEL
LIN {X 0,Y 177.109,Z 241.369,A -85,B 0,C 180,E1 -25361.49,E2 -25361.49} C_VEL
LIN {X 0,Y 175.944,Z 238.304,A -85,B 0,C 180,E1 -25365.616,E2 -25365.616} C_VEL
LIN {X 0,Y 175.356,Z 237.887,A -85,B 0,C 180,E1 -25370.774,E2 -25370.774} C_VEL
LIN {X 0,Y 176.388,Z 238.529,A -85,B 0,C 180,E1 -25376.468,E2 -25376.468} C_VEL
LIN {X 0,Y 177.813,Z 241.904,A -85,B 0,C 180,E1 -25380.49,E2 -25380.49} C_VEL
LIN {X 0,Y 178.868,Z 243.255,A -85,B 0,C 180,E1 -25382.349,E2 -25382.349} C_VEL
LIN {X 0,Y 180.984,Z 246.958,A -85,B 0,C 180,E1 -25385.546,E2 -25385.546} C_VEL
LIN {X 0,Y 183.84,Z 252.091,A -85,B 0,C 180,E1 -25389.001,E2 -25389.001} C_VEL
LIN {X 0,Y 187.804,Z 259.465,A -85,B 0,C 180,E1 -25392.81,E2 -25392.81} C_VEL
LIN {X 0,Y 190.059,Z 264.083,A -85,B 0,C 180,E1 -25394.706,E2 -25394.706} C_VEL
LIN {X 0,Y 188.096,Z 282.525,A -85,B 0,C 180,E1 -25395.344,E2 -25395.344} C_VEL
LIN {X 0,Y 185.665,Z 294.967,A -85,B 0,C 180,E1 -25395.997,E2 -25395.997} C_VEL
LIN {X 0,Y 182.303,Z 307.081,A -85,B 0,C 180,E1 -25396.951,E2 -25396.951} C_VEL
LIN {X 0,Y 177.704,Z 319.565,A -85,B 0,C 180,E1 -25398.345,E2 -25398.345} C_VEL
LIN {X 0,Y 172.767,Z 330.112,A -85,B 0,C 180,E1 -25399.873,E2 -25399.873} C_VEL
LIN {X 0,Y 167.379,Z 339.769,A -85,B 0,C 180,E1 -25401.721,E2 -25401.721} C_VEL
LIN {X 0,Y 161.477,Z 348.682,A -85,B 0,C 180,E1 -25403.938,E2 -25403.938} C_VEL
LIN {X 0,Y 154.949,Z 357.113,A -85,B 0,C 180,E1 -25406.723,E2 -25406.723} C_VEL
LIN {X 0,Y 148.183,Z 364.612,A -85,B 0,C 180,E1 -25410.054,E2 -25410.054} C_VEL
LIN {X 0,Y 142.771,Z 369.844,A -85,B 0,C 180,E1 -25413.193,E2 -25413.193} C_VEL
LIN {X 0,Y 136.939,Z 374.83,A -85,B 0,C 180,E1 -25417.301,E2 -25417.301} C_VEL
LIN {X 0,Y 131.823,Z 378.53,A -85,B 0,C 180,E1 -25421.721,E2 -25421.721} C_VEL
LIN {X 0,Y 128.462,Z 380.545,A -85,B 0,C 180,E1 -25425.331,E2 -25425.331} C_VEL
LIN {X 0,Y 124.113,Z 382.514,A -85,B 0,C 180,E1 -25431.473,E2 -25431.473} C_VEL
LIN {X 0,Y 122.341,Z 382.882,A -85,B 0,C 180,E1 -25434.939,E2 -25434.939} C_VEL
LIN {X 0,Y 120.087,Z 382.442,A -85,B 0,C 180,E1 -25441.382,E2 -25441.382} C_VEL
LIN {X 0,Y 119.252,Z 381.349,A -85,B 0,C 180,E1 -25445.636,E2 -25445.636} C_VEL
LIN {X 0,Y 118.974,Z 379.117,A -85,B 0,C 180,E1 -25450.929,E2 -25450.929} C_VEL
LIN {X 0,Y 119.416,Z 375.711,A -85,B 0,C 180,E1 -25456.385,E2 -25456.385} C_VEL
LIN {X 0,Y 120.632,Z 370.816,A -85,B 0,C 180,E1 -25462.048,E2 -25462.048} C_VEL
LIN {X 0,Y 122.53,Z 364.483,A -85,B 0,C 180,E1 -25467.535,E2 -25467.535} C_VEL
LIN {X 0,Y 124.955,Z 357.057,A -85,B 0,C 180,E1 -25472.418,E2 -25472.418} C_VEL
LIN {X 0,Y 128.126,Z 347.82,A -85,B 0,C 180,E1 -25477.09,E2 -25477.09} C_VEL
LIN {X 0,Y 131.368,Z 338.23,A -85,B 0,C 180,E1 -25480.793,E2 -25480.793} C_VEL
LIN {X 0,Y 134.584,Z 327.565,A -85,B 0,C 180,E1 -25483.977,E2 -25483.977} C_VEL
LIN {X 0,Y 137.801,Z 315.66,A -85,B 0,C 180,E1 -25486.672,E2 -25486.672} C_VEL
LIN {X 0,Y 140.239,Z 304.132,A -85,B 0,C 180,E1 -25488.633,E2 -25488.633} C_VEL
LIN {X 0,Y 142.488,Z 290.613,A -85,B 0,C 180,E1 -25490.264,E2 -25490.264} C_VEL
LIN {X 0,Y 143.931,Z 278.067,A -85,B 0,C 180,E1 -25491.245,E2 -25491.245} C_VEL
LIN {X 0,Y 147.068,Z 228.496,A -85,B 0,C 180,E1 -25493.48,E2 -25493.48} C_VEL
LIN {X 0,Y 140.468,Z 213.989,A -85,B 0,C 180,E1 -25496.403,E2 -25496.403} C_VEL
LIN {X 0,Y 134.105,Z 202.584,A -85,B 0,C 180,E1 -25499.439,E2 -25499.439} C_VEL
LIN {X 0,Y 129.87,Z 195.825,A -85,B 0,C 180,E1 -25501.619,E2 -25501.619} C_VEL
LIN {X 0,Y 127.309,Z 192.037,A -85,B 0,C 180,E1 -25503.025,E2 -25503.025} C_VEL
LIN {X 0,Y 125.149,Z 188.659,A -85,B 0,C 180,E1 -25504.3,E2 -25504.3} C_VEL
LIN {X 0,Y 122.622,Z 185.661,A -85,B 0,C 180,E1 -25505.806,E2 -25505.806} C_VEL
LIN {X 0,Y 121.878,Z 183.273,A -85,B 0,C 180,E1 -25506.533,E2 -25506.533} C_VEL
LIN {X 0,Y 121.861,Z 183.305,A -85,B 0,C 180,E1 -25511.435,E2 -25511.435} C_VEL
LIN {X 0,Y 121.844,Z 183.268,A -85,B 0,C 180,E1 -25518.578,E2 -25518.578} C_VEL
LIN {X 0,Y 121.906,Z 183.291,A -85,B 0,C 180,E1 -25524.797,E2 -25524.797} C_VEL
LIN {X 0,Y 121.904,Z 183.235,A -85,B 0,C 180,E1 -25529.859,E2 -25529.859} C_VEL
LIN {X 0,Y 121.979,Z 183.289,A -85,B 0,C 180,E1 -25537.202,E2 -25537.202} C_VEL
LIN {X 0,Y 122.058,Z 183.265,A -85,B 0,C 180,E1 -25543.27,E2 -25543.27} C_VEL
LIN {X 0,Y 122.288,Z 183.253,A -85,B 0,C 180,E1 -25547.695,E2 -25547.695} C_VEL
LIN {X 0,Y 122.391,Z 183.224,A -85,B 0,C 180,E1 -25550.082,E2 -25550.082} C_VEL
LIN {X 0,Y 122.56,Z 183.218,A -85,B 0,C 180,E1 -25556.714,E2 -25556.714} C_VEL
LIN {X 0,Y 123.023,Z 183.145,A -85,B 0,C 180,E1 -25560.002,E2 -25560.002} C_VEL
LIN {X 0,Y 122.408,Z 183.227,A -85,B 0,C 180,E1 -25566.596,E2 -25566.596} C_VEL
LIN {X 0,Y 122.393,Z 183.231,A -85,B 0,C 180,E1 -25569.921,E2 -25569.921} C_VEL
LIN {X 0,Y 122.19,Z 183.263,A -85,B 0,C 180,E1 -25573.303,E2 -25573.303} C_VEL
LIN {X 0,Y 121.993,Z 183.29,A -85,B 0,C 180,E1 -25580.224,E2 -25580.224} C_VEL
LIN {X 0,Y 121.949,Z 183.295,A -85,B 0,C 180,E1 -25583.794,E2 -25583.794} C_VEL
LIN {X 0,Y 121.93,Z 183.296,A -85,B 0,C 180,E1 -25590.162,E2 -25590.162} C_VEL
LIN {X 0,Y 121.934,Z 183.298,A -85,B 0,C 180,E1 -25593.078,E2 -25593.078} C_VEL
LIN {X 0,Y 122.817,Z 185.999,A -85,B 0,C 180,E1 -25593.791,E2 -25593.791} C_VEL
LIN {X 0,Y 125.299,Z 188.999,A -85,B 0,C 180,E1 -25595.267,E2 -25595.267} C_VEL
LIN {X 0,Y 127.411,Z 192.196,A -85,B 0,C 180,E1 -25596.504,E2 -25596.504} C_VEL
LIN {X 0,Y 133.135,Z 200.979,A -85,B 0,C 180,E1 -25599.553,E2 -25599.553} C_VEL
LIN {X 0,Y 135.664,Z 205.735,A -85,B 0,C 180,E1 -25600.848,E2 -25600.848} C_VEL
LIN {X 0,Y 140.683,Z 217.63,A -85,B 0,C 180,E1 -25603.387,E2 -25603.387} C_VEL
LIN {X 0,Y 144.99,Z 230.326,A -85,B 0,C 180,E1 -25605.518,E2 -25605.518} C_VEL
LIN {X 0,Y 145.437,Z 233.338,A -85,B 0,C 180,E1 -25605.834,E2 -25605.834} C_VEL
LIN {X 0,Y 146.326,Z 245.119,A -85,B 0,C 180,E1 -25606.806,E2 -25606.806} C_VEL
LIN {X 0,Y 143.542,Z 287.672,A -85,B 0,C 180,E1 -25608.737,E2 -25608.737} C_VEL
LIN {X 0,Y 141.836,Z 300.962,A -85,B 0,C 180,E1 -25609.8,E2 -25609.8} C_VEL
LIN {X 0,Y 139.612,Z 312.968,A -85,B 0,C 180,E1 -25611.236,E2 -25611.236} C_VEL
LIN {X 0,Y 137.19,Z 323.584,A -85,B 0,C 180,E1 -25612.991,E2 -25612.991} C_VEL
LIN {X 0,Y 133.817,Z 335.582,A -85,B 0,C 180,E1 -25615.626,E2 -25615.626} C_VEL
LIN {X 0,Y 130.468,Z 346.296,A -85,B 0,C 180,E1 -25618.769,E2 -25618.769} C_VEL
LIN {X 0,Y 127.78,Z 354.411,A -85,B 0,C 180,E1 -25621.813,E2 -25621.813} C_VEL
LIN {X 0,Y 124.886,Z 363.099,A -85,B 0,C 180,E1 -25625.92,E2 -25625.92} C_VEL
LIN {X 0,Y 122.773,Z 369.755,A -85,B 0,C 180,E1 -25629.911,E2 -25629.911} C_VEL
LIN {X 0,Y 120.85,Z 376.266,A -85,B 0,C 180,E1 -25634.829,E2 -25634.829} C_VEL
LIN {X 0,Y 119.829,Z 381.412,A -85,B 0,C 180,E1 -25639.865,E2 -25639.865} C_VEL
LIN {X 0,Y 119.406,Z 385.365,A -85,B 0,C 180,E1 -25644.934,E2 -25644.934} C_VEL
LIN {X 0,Y 119.568,Z 388.248,A -85,B 0,C 180,E1 -25649.999,E2 -25649.999} C_VEL
LIN {X 0,Y 119.42,Z 389.562,A -85,B 0,C 180,E1 -25653.373,E2 -25653.373} C_VEL
LIN {X 0,Y 119.824,Z 391.011,A -85,B 0,C 180,E1 -25660.134,E2 -25660.134} C_VEL
LIN {X 0,Y 120.525,Z 391.167,A -85,B 0,C 180,E1 -25663.488,E2 -25663.488} C_VEL
LIN {X 0,Y 123.071,Z 390.277,A -85,B 0,C 180,E1 -25670.037,E2 -25670.037} C_VEL
LIN {X 0,Y 127.376,Z 387.879,A -85,B 0,C 180,E1 -25676.193,E2 -25676.193} C_VEL
LIN {X 0,Y 131.541,Z 384.99,A -85,B 0,C 180,E1 -25680.502,E2 -25680.502} C_VEL
LIN {X 0,Y 136.227,Z 381.116,A -85,B 0,C 180,E1 -25684.575,E2 -25684.575} C_VEL
LIN {X 0,Y 140.954,Z 376.884,A -85,B 0,C 180,E1 -25687.821,E2 -25687.821} C_VEL
LIN {X 0,Y 142.34,Z 375.11,A -85,B 0,C 180,E1 -25689.158,E2 -25689.158} C_VEL
LIN {X 0,Y 144.3,Z 369.199,A -85,B 0,C 180,E1 -25693.957,E2 -25693.957} C_VEL
LIN {X 0,Y 145.984,Z 367,A -85,B 0,C 180,E1 -25695.088,E2 -25695.088} C_VEL
LIN {X 0,Y 152.064,Z 359.97,A -85,B 0,C 180,E1 -25697.687,E2 -25697.687} C_VEL
LIN {X 0,Y 158.294,Z 351.771,A -85,B 0,C 180,E1 -25699.985,E2 -25699.985} C_VEL
LIN {X 0,Y 164.863,Z 341.775,A -85,B 0,C 180,E1 -25702.059,E2 -25702.059} C_VEL
LIN {X 0,Y 170.308,Z 331.906,A -85,B 0,C 180,E1 -25703.581,E2 -25703.581} C_VEL
LIN {X 0,Y 175.901,Z 319.48,A -85,B 0,C 180,E1 -25704.991,E2 -25704.991} C_VEL
LIN {X 0,Y 180.245,Z 307.045,A -85,B 0,C 180,E1 -25706.002,E2 -25706.002} C_VEL
LIN {X 0,Y 183.636,Z 293.299,A -85,B 0,C 180,E1 -25706.765,E2 -25706.765} C_VEL
LIN {X 0,Y 185.6,Z 279.909,A -85,B 0,C 180,E1 -25707.29,E2 -25707.29} C_VEL
LIN {X 0,Y 186.194,Z 273.291,A -85,B 0,C 180,E1 -25707.518,E2 -25707.518} C_VEL
LIN {X 0,Y 183.568,Z 265.87,A -85,B 0,C 180,E1 -25710.209,E2 -25710.209} C_VEL
LIN {X 0,Y 181.107,Z 259.44,A -85,B 0,C 180,E1 -25713.15,E2 -25713.15} C_VEL
LIN {X 0,Y 178.743,Z 253.838,A -85,B 0,C 180,E1 -25716.542,E2 -25716.542} C_VEL
LIN {X 0,Y 176.957,Z 249.885,A -85,B 0,C 180,E1 -25719.769,E2 -25719.769} C_VEL
LIN {X 0,Y 174.938,Z 245.285,A -85,B 0,C 180,E1 -25726.051,E2 -25726.051} C_VEL
LIN {X 0,Y 174.68,Z 245.022,A -85,B 0,C 180,E1 -25733.066,E2 -25733.066} C_VEL
LIN {X 0,Y 175.344,Z 245.467,A -85,B 0,C 180,E1 -25736.018,E2 -25736.018} C_VEL
LIN {X 0,Y 176.761,Z 248.904,A -85,B 0,C 180,E1 -25740.246,E2 -25740.246} C_VEL
LIN {X 0,Y 177.675,Z 250.195,A -85,B 0,C 180,E1 -25741.947,E2 -25741.947} C_VEL
LIN {X 0,Y 179.556,Z 253.739,A -85,B 0,C 180,E1 -25744.957,E2 -25744.957} C_VEL
LIN {X 0,Y 182.06,Z 258.418,A -85,B 0,C 180,E1 -25748.17,E2 -25748.17} C_VEL
LIN {X 0,Y 185.679,Z 265.576,A -85,B 0,C 180,E1 -25751.913,E2 -25751.913} C_VEL
LIN {X 0,Y 186.667,Z 267.716,A -85,B 0,C 180,E1 -25752.822,E2 -25752.822} C_VEL
LIN {X 0,Y 185.996,Z 275.49,A -85,B 0,C 180,E1 -25753.127,E2 -25753.127} C_VEL
LIN {X 0,Y 183.846,Z 289.221,A -85,B 0,C 180,E1 -25753.677,E2 -25753.677} C_VEL
LIN {X 0,Y 180.966,Z 301.076,A -85,B 0,C 180,E1 -25754.425,E2 -25754.425} C_VEL
LIN {X 0,Y 176.913,Z 313.353,A -85,B 0,C 180,E1 -25755.561,E2 -25755.561} C_VEL
LIN {X 0,Y 171.861,Z 325.083,A -85,B 0,C 180,E1 -25757.006,E2 -25757.006} C_VEL
LIN {X 0,Y 166.092,Z 335.901,A -85,B 0,C 180,E1 -25758.778,E2 -25758.778} C_VEL
LIN {X 0,Y 159.909,Z 345.505,A -85,B 0,C 180,E1 -25760.892,E2 -25760.892} C_VEL
LIN {X 0,Y 153.247,Z 354.3,A -85,B 0,C 180,E1 -25763.478,E2 -25763.478} C_VEL
LIN {X 0,Y 145.708,Z 362.736,A -85,B 0,C 180,E1 -25766.834,E2 -25766.834} C_VEL
LIN {X 0,Y 138.701,Z 369.325,A -85,B 0,C 180,E1 -25770.527,E2 -25770.527} C_VEL
LIN {X 0,Y 132.402,Z 374.468,A -85,B 0,C 180,E1 -25774.639,E2 -25774.639} C_VEL
LIN {X 0,Y 126.802,Z 378.326,A -85,B 0,C 180,E1 -25779.109,E2 -25779.109} C_VEL
LIN {X 0,Y 122.397,Z 380.835,A -85,B 0,C 180,E1 -25783.551,E2 -25783.551} C_VEL
LIN {X 0,Y 118.165,Z 382.623,A -85,B 0,C 180,E1 -25789.139,E2 -25789.139} C_VEL
LIN {X 0,Y 116.102,Z 383.125,A -85,B 0,C 180,E1 -25792.748,E2 -25792.748} C_VEL
LIN {X 0,Y 114.443,Z 383.138,A -85,B 0,C 180,E1 -25796.448,E2 -25796.448} C_VEL
LIN {X 0,Y 113.199,Z 382.705,A -85,B 0,C 180,E1 -25800.361,E2 -25800.361} C_VEL
LIN {X 0,Y 112.394,Z 381.875,A -85,B 0,C 180,E1 -25804.043,E2 -25804.043} C_VEL
LIN {X 0,Y 111.892,Z 379.414,A -85,B 0,C 180,E1 -25810.411,E2 -25810.411} C_VEL
LIN {X 0,Y 112.186,Z 376.529,A -85,B 0,C 180,E1 -25815.488,E2 -25815.488} C_VEL
LIN {X 0,Y 113.204,Z 372.342,A -85,B 0,C 180,E1 -25820.93,E2 -25820.93} C_VEL
LIN {X 0,Y 114.868,Z 366.68,A -85,B 0,C 180,E1 -25826.493,E2 -25826.493} C_VEL
LIN {X 0,Y 117.165,Z 359.768,A -85,B 0,C 180,E1 -25831.719,E2 -25831.719} C_VEL
LIN {X 0,Y 120.344,Z 351.147,A -85,B 0,C 180,E1 -25836.708,E2 -25836.708} C_VEL
LIN {X 0,Y 123.867,Z 341.239,A -85,B 0,C 180,E1 -25841.041,E2 -25841.041} C_VEL
LIN {X 0,Y 127.189,Z 331.255,A -85,B 0,C 180,E1 -25844.399,E2 -25844.399} C_VEL
LIN {X 0,Y 130.424,Z 320.253,A -85,B 0,C 180,E1 -25847.241,E2 -25847.241} C_VEL
LIN {X 0,Y 133.202,Z 308.915,A -85,B 0,C 180,E1 -25849.455,E2 -25849.455} C_VEL
LIN {X 0,Y 135.73,Z 296.262,A -85,B 0,C 180,E1 -25851.252,E2 -25851.252} C_VEL
LIN {X 0,Y 137.499,Z 283.344,A -85,B 0,C 180,E1 -25852.522,E2 -25852.522} C_VEL
LIN {X 0,Y 138.787,Z 267.993,A -85,B 0,C 180,E1 -25853.374,E2 -25853.374} C_VEL
